arTonDelay[01](IN:=, PT:=T#1S , Q=> , ET=> );
arTonDelay[02](IN:= , PT:=T#1S , Q=> , ET=> );//注液延时使用
arTonDelay[03](IN:= , PT:=T#10S , Q=> , ET=> );
arTonDelay[04](IN:= , PT:=T#0.1S , Q=> , ET=> );
arTonDelay[05](IN:= , PT:=T#0.1S , Q=> , ET=> );
arTonDelay[06](IN:= , PT:=T#0.1S , Q=> , ET=> );
arTonDelay[07](IN:=NOT  fbXAxisMove.xbusy, PT:=T#0.1S , Q=> , ET=> );//TipAuto使用
arTonDelay[08](IN:=NOT  fbYAxisMove.xbusy , PT:=T#0.1S , Q=> , ET=> );//TipAuto使用
arTonDelay[09](IN:= NOT  fbZAxisMove.xbusy, PT:=T#0.1S , Q=> , ET=> );//TipAuto使用
arTonDelay[10](IN:= NOT fbStirAxis.xbusy, PT:=T#0.1S , Q=> , ET=> );//TipAuto使用
END_ACTION

ACTION FlowAuto:

//-----------------------------------------初始化是否完成判断----------------------------------------------
IF NOT station.xInitDone 
THEN
 	station.iStepAuto:=0;
 	station.xDone:=FALSE;
	station.xRunningOffProhibit := FALSE ;//运行中信号Off禁止
ELSIF station.xRunning OR  
(tsModuleProcess[bXCounter+1].xProcessStarted AND  NOT tsModuleProcess[bXCounter+1].xProcessCompleted)//注液流程
THEN
//-----------------------------------------动作步骤--------------------------------------------------------
CASE station.iStepAuto OF	  
	0: //----Home Step，等待启动----
		IF station.xDisabled 
			AND station.xCanRun 
			AND NOT fbMachine[1].xStopped 
			AND NOT station.xSingleRunning 
		THEN
			station.xDone:=TRUE;
		END_IF
		
		IF  station.xSingleRunning 
			OR station.xCanRun 
			AND NOT station.xDone 
			AND NOT station.xDisabled 
			AND NOT fbMachine[1].xStopped
		THEN
			station.xCycleEnable:=TRUE;
			station.xDone:= FALSE;  
			station.iStepAuto:= 10;
		END_IF
    10: //复位数据 
			FOR i:=1 TO gc_ModuleProNo BY 1 DO
				MEMSET(ADR(tsModuleProcess[i]),0,SIZEOF(tsModuleProcess[i]));
			END_FOR
			station.iStepAuto:=15;
	
	 15://程序分类选择
			IF NOT   fbMachine[1].xTryRun THEN
					 IF  station.xSingleRunning AND stCalibration.xNeedCalibration THEN//进入校准程序
							stCalibration.xWindowsTrigger:=TRUE;
							station.iStepAuto:=1000;
					 ELSE //进入正常程序
						 station.iStepAuto:=20;
					 END_IF
		 ELSE
					 station.iStepAuto:=20;
			END_IF
	20:////Restore_after_Estop_Process1 上载数据流程
			IF  station.xSingleRunning THEN  //OR fbMachine[1].xTryRun THEN
					station.iStepAuto :=45; 
			ELSIF tsModuleProcess[1].xProcessNotStarted AND NOT  tsModuleProcess[1].xProcessStarted THEN
					station.iStepAuto :=21; (*process not started*)
			ELSIF  tsModuleProcess[1].xProcessStarted AND NOT  tsModuleProcess[1].xProcessCompleted THEN
				 station.iStepAuto :=21 ;(*process started*)
			ELSIF  tsModuleProcess[1].xProcessCompleted AND NOT tsModuleProcess[1].xQDataCompleted  THEN
					station.iStepAuto :=30  ;(*process completed*)
			ELSIF tsModuleProcess[1].xQDataCompleted THEN
					station.iStepAuto :=30;(*Qdata completed *)
			ELSE
					station.iStepAuto :=21; 
			END_IF	
	21:	
			tsModuleProcess[1].xProcessNotStarted :=TRUE;
			station.iStepAuto :=25;
	25://数据load 
		tsModuleProcess[1].xProcessStarted:=TRUE;
		MEMCPY(ADR(arProcessDataStation[1]),ADR(arMainlineFixtureData[arCurFixtureNumStation[3]]),SIZEOF(arMainlineFixtureData[arCurFixtureNumStation[3]]));
		MEMCPY(ADR(arProcessDataStation[2]),ADR(arMainlineFixtureData[arCurFixtureNumStation[4]]),SIZEOF(arMainlineFixtureData[arCurFixtureNumStation[4]]));
		tsModuleProcess[1].xProcessCompleted:=TRUE;	
		tsModuleProcess[1].xQDataCompleted:=TRUE;	
		station.iStepAuto:= 30;
	/////产品流程开始	
	30: //判断产品状态
			 IF NOT  fbMachine[1].xTryRun THEN
					IF    station.xEmptyDone THEN //清料完成
							 station.iStepAuto:=998;
					ELSIF     //清料程序执行条件
							 arProcessDataStation[1].stProduct.xEmptying AND 
							 arProcessDataStation[2].stProduct.xEmptying AND 
							 NOT xSensorReached[1] AND  NOT   xSensorReached[2] THEN
										station.xEmptying :=TRUE;	
									  station.iStepAuto:= 2000; 
					ELSIF //第一站由于需要增加节拍增加了并行程序，所以写入请料的时机不好把控
					 			//在本站增加此条件以修正请料信号的位置
							 arProcessDataStation[1].stProduct.xEmptying AND 
							 arProcessDataStation[2].stProduct.xEmptying AND 
							  xSensorReached[1] AND  xSensorReached[2] THEN
										arProcessDataStation[1].stProduct.xEmptying :=FALSE; 		
								    arProcessDataStation[2].stProduct.xEmptying :=FALSE;
										arProcessDataStation[1].xMaterialOnOff :=TRUE; 		
								    arProcessDataStation[2].xMaterialOnOff :=TRUE;  
									  station.iStepAuto:= 40;
					ELSIF   (arProcessDataStation[1].xMaterialOnOff   AND
								  arProcessDataStation[2].xMaterialOnOff ) OR
									(xSensorReached[1] AND   xSensorReached[2])  THEN
										station.iStepAuto:= 40;  
					ELSIF		 NOT arProcessDataStation[1].xMaterialOnOff   AND
								   NOT arProcessDataStation[2].xMaterialOnOff  AND 
									 NOT xSensorReached[1]  AND  NOT xSensorReached[2]  THEN
									station.iStepAuto:= 998;
					END_IF
			 ELSE
					 station.iStepAuto:= 40;
			 END_IF
	40://写入NOK按钮
		IF   arManualNOKHmiButton[2]  AND NOT station.xSingleRunning THEN
			station.iStepAuto:=155;
			arManualNOKHmiButton[2]:=FALSE;
		ELSE
			 station.iStepAuto:=45;
		END_IF
	
	//////产品流程开始
	45://循环开始次数为1，总循环为2
			 bXCounter:=1;
	    station.iStepAuto:= 50;

	50:////Restore_after_Estop_Process1/2 注液流程1/2
			IF  station.xSingleRunning  OR fbMachine[1].xTryRun THEN
					station.iStepAuto :=80; 
			ELSIF tsModuleProcess[bXCounter+1].xProcessNotStarted AND NOT  tsModuleProcess[bXCounter+1].xProcessStarted THEN
					station.iStepAuto :=100; (*process not started*)
			ELSIF  tsModuleProcess[bXCounter+1].xProcessStarted AND NOT  tsModuleProcess[bXCounter+1].xProcessCompleted THEN
				 station.iStepAuto :=155 ;(*process started*)
			ELSIF  tsModuleProcess[bXCounter+1].xProcessCompleted AND NOT tsModuleProcess[bXCounter+1].xQDataCompleted  THEN
					station.iStepAuto :=150  ;(*process completed*)
			ELSIF tsModuleProcess[bXCounter+1].xQDataCompleted THEN
					station.iStepAuto :=160;(*Qdata completed *)
			ELSE
					station.iStepAuto :=80; 
			END_IF

	80://流程未开始
			 tsModuleProcess[bXCounter+1].xProcessNotStarted:=TRUE;
		 		station.iStepAuto:= 90;
	90://水平调整气缸伸出
		IF  iBoxChoose =1 THEN
			(*上层水平调整气缸*)
			fbHOZAdjustCyl_1.xAuto :=TRUE;
		//	fbHOZAdjustCyl_2.xAuto :=TRUE;
			IF  fbHOZAdjustCyl_1.xWP_Delay THEN// AND fbHOZAdjustCyl_2.xWP_Delay  THEN
					station.iStepAuto:= 100;
			END_IF
		ELSIF  iBoxChoose= 2 THEN
			(*下层水平调整气缸*)
			fbHOZAdjustCyl_3.xAuto :=TRUE;
			//fbHOZAdjustCyl_4.xAuto :=TRUE;
			IF  fbHOZAdjustCyl_3.xWP_Delay  THEN//AND fbHOZAdjustCyl_4.xWP_Delay  THEN
					station.iStepAuto:= 100;
			END_IF
		END_IF	 
	100://XY轴去注液位置1、2
			fbXAxisMove.xMoveAuto[bXCounter+1]:=TRUE;
			fbYAxisMove.xMoveAuto[bXCounter+1]:=TRUE;
			IF fbXAxisMove.xMoveInPos[bXCounter+1]  AND fbYAxisMove.xMoveInPos[bXCounter+1]  THEN
				station.iStepAuto:=110;	
			END_IF
	110:	//防滴液气缸伸出
		fbROTCyl.xAuto:=TRUE;
		IF fbROTCyl.xWP_Delay THEN
			station.iStepAuto:=120;	
		END_IF
	120://Z轴下降去注液位置
		   fbZAxisMove.xMoveAuto[2]:=TRUE;
		IF  fbZAxisMove.xMoveInPos[2] THEN
			station.iStepAuto:=125;
		END_IF
	125://屏蔽注液
			FOR i:=1 TO  12 BY 1 DO
					arxPushBusy[i]:=FALSE;
		 END_FOR
			IF   axBypassSignal[2] OR fbMachine[1].xTryRun THEN
				station.iStepAuto:=145;
			ELSE
				station.iStepAuto:=130;
			END_IF
	130://开始注液
		  tsModuleProcess[bXCounter+1].xProcessStarted:=TRUE;
		 FOR i:=1 TO  12 BY 1 DO
						fbEasyPumps[i].stDeviceOpe.xPush_Auto[1]:=TRUE;
						IF  fbEasyPumps[i].xQBusy THEN
						 		arxPushBusy[i]:=TRUE;
						END_IF
		 END_FOR
		 	FOR   i :=1 TO 12 BY  1  DO
			 			IF NOT  arxPushBusy[i] THEN
						 		EXIT;
						ELSIF i =12 THEN
						 	  station.iStepAuto:=140;	
					  END_IF
			END_FOR
	140://注液结束
					arTonDelay[02](IN:=FALSE );
					 IF   	fbEasyPumps[1].xQDone AND
									fbEasyPumps[2].xQDone AND
									fbEasyPumps[3].xQDone AND
								  fbEasyPumps[4].xQDone AND
									fbEasyPumps[5].xQDone AND
									fbEasyPumps[6].xQDone AND
									fbEasyPumps[7].xQDone AND
								  fbEasyPumps[8].xQDone AND
									fbEasyPumps[9].xQDone AND
									fbEasyPumps[10].xQDone AND
									fbEasyPumps[11].xQDone AND
								  fbEasyPumps[12].xQDone THEN						
								 station.iStepAuto:=145;	
					 END_IF
	145://注液完成
		tsModuleProcess[bXCounter+1].xProcessCompleted:=TRUE;
		 station.iStepAuto:=150;	
	150://写入结果
				arProcessDataStation[bXCounter].xMaterialOnOff:=TRUE;
				arProcessDataStation[bXCounter].stProduct.xlidInjecting_OK:=TRUE;
				arProcessDataStation[bXCounter].stProduct.xlidInjecting_NOK:=FALSE;	
			 tsModuleProcess[bXCounter].xQDataCompleted:=TRUE;
			 station.iStepAuto:=160;
	155://注液失败
				arProcessDataStation[bXCounter].xMaterialOnOff:=TRUE;
				arProcessDataStation[bXCounter].stProduct.xlidInjecting_OK:=FALSE;
				arProcessDataStation[bXCounter].stProduct.xlidInjecting_NOK:=TRUE;	
				station.iStepAuto:=160;
	160://Z轴上升
		  fbZAxisMove.xMoveAuto[1]:=TRUE;
		IF  fbZAxisMove.xMoveInPos[1] THEN
			station.iStepAuto:=170;
		END_IF
	170://防滴漏气缸收回
		fbROTCyl.xAuto:=FALSE;
		IF fbROTCyl.xHP_Delay THEN
			station.iStepAuto:=180;	
		END_IF
	180://循环+1
		 	bXCounter:=bXCounter +1 ;
			station.iStepAuto:=190;
	190://检查循环次数
			IF   bXCounter<=2 THEN
				station.iStepAuto:=50;
			ELSE
				station.iStepAuto:=200;
			END_IF
	200://水平调整气缸收回
			IF  iBoxChoose =1 THEN
			(*上层水平调整气缸*)
			fbHOZAdjustCyl_1.xAuto :=FALSE;
		//	fbHOZAdjustCyl_2.xAuto :=FALSE;
			IF  fbHOZAdjustCyl_1.xHP_Delay THEN  // AND fbHOZAdjustCyl_2.xHP_Delay  THEN
					station.iStepAuto:= 210;
			END_IF
		ELSIF  iBoxChoose= 2 THEN
			(*下层水平调整气缸*)
			fbHOZAdjustCyl_3.xAuto :=FALSE;
		//	fbHOZAdjustCyl_4.xAuto :=FALSE;
			IF  fbHOZAdjustCyl_3.xHP_Delay  THEN // AND fbHOZAdjustCyl_4.xHP_Delay  THEN
					station.iStepAuto:= 210;
			END_IF
		END_IF
	210:////产品流程结束	
		station.iStepAuto:= 220;
		
	220://Restore_after_Estop_Process4 数据传输 
			IF  station.xSingleRunning THEN // OR fbMachine[1].xTryRun THEN
					station.iStepAuto :=998; 
			ELSIF tsModuleProcess[4].xProcessNotStarted AND NOT  tsModuleProcess[4].xProcessStarted THEN
					station.iStepAuto :=550; (*process not started*)
			ELSIF  tsModuleProcess[4].xProcessStarted AND NOT  tsModuleProcess[4].xProcessCompleted THEN
				 station.iStepAuto :=550 ;(*process started*)
			ELSIF  tsModuleProcess[4].xProcessCompleted AND NOT tsModuleProcess[4].xQDataCompleted  THEN
					station.iStepAuto :=560  ;(*process completed*)
			ELSIF tsModuleProcess[4].xQDataCompleted THEN
					station.iStepAuto :=999;(*Qdata completed *)
			ELSE
					station.iStepAuto :=550; 
			END_IF
	550://数据unload
			tsModuleProcess[4].xProcessNotStarted :=TRUE;
			tsModuleProcess[4].xProcessStarted :=TRUE;
			MEMCPY(ADR(arMainlineFixtureData[arCurFixtureNumStation[3]]),ADR(arProcessDataStation[1]),SIZEOF(arProcessDataStation[1]));
			MEMCPY(ADR(arMainlineFixtureData[arCurFixtureNumStation[4]]),ADR(arProcessDataStation[2]),SIZEOF(arProcessDataStation[2]));
			station.iStepAuto:= 560;
		
	560:
			tsModuleProcess[4].xProcessCompleted :=TRUE;
			station.iStepAuto:= 570;
 	570://本地数据清除
			//MEMSET(ADR(arProcessDataStation[1]),0,SIZEOF(arProcessDataStation[1]));
			//MEMSET(ADR(arProcessDataStation[2]),0,SIZEOF(arProcessDataStation[2]));
			tsModuleProcess[4].xQDataCompleted:=TRUE;
			arManualNOKHmiButton[2]:=FALSE;
			station.iStepAuto:= 998;
		
	998://----Single Run Finish----
		station.iStepAuto :=999;
		IF NOT station.xSingleContinuousRun THEN
			station.xSingleRunFlag:=FALSE;
		END_IF
		station.xCycleEnable:=FALSE;	
		station.xDone:=TRUE;
		
	999://XY伺服回参考位置
			fbXAxisMove.xMoveAuto[1]:=TRUE;
			fbYAxisMove.xMoveAuto[1]:=TRUE;
			IF fbXAxisMove.xMoveInPos[1]  AND fbYAxisMove.xMoveInPos[1]  THEN
				station.iStepAuto:=0;	
			END_IF
	{region "蠕动泵校准程序"}
	1000://切换窗口
			stCalibration.xWindowsTrigger:=TRUE;
			iCalibStep:=station.iStepAuto;
			station.iStepAuto:=1010;
	1010://等待人工安装好校准工装,
		 stCalibration.strCalibHmi:='Please Load Calibration Tool and then press Start Button ';
		IF    stCalibration.xStartButtonHmi THEN
			station.iStepAuto:=1020;
		END_IF
			 	iCalibStep:=station.iStepAuto;
	1020://开始循环
		 	FOR i:=1 TO 12 BY 1 DO
				 IF 	NOT arxRudongPumpCalibBypass[i] THEN
						 stCalibration.iYCounter:=i;
						 EXIT;
				 END_IF
			END_FOR
			stCalibration.iXCounter:=1;
			//stCalibration.iYCounter:=1;
			iCalibStep:=station.iStepAuto;
			station.iStepAuto:=1030;
		{region "初始化开始"}	
	1030://初始化蠕动泵
			stCalibration.strCalibHmi:='All RuDongPump is initing，please Wait it';
			station.iStepAuto:=station.iStepAuto +1;
			iCalibStep:=station.iStepAuto;
	1031://蠕动泵初始化开始
				 FOR i:=1 TO  12 BY 1 DO
						fbEasyPumps[i].stDeviceOpe.xStop_auto:=TRUE;
						IF	NOT fbEasyPumps[i].xQBusy  THEN
								EXIT;
						ELSIF   i =12 THEN
									iCalibStep:=station.iStepAuto;
									station.iStepAuto:=station.iStepAuto +1;		
					 	END_IF						
				 END_FOR
	1032://蠕动泵停
					iCalibStep:=station.iStepAuto;
					IF   fbEasyPumps[1].xQDone AND 
							 fbEasyPumps[2].xQDone AND 
							 fbEasyPumps[3].xQDone AND 
							 fbEasyPumps[4].xQDone AND 
							 fbEasyPumps[5].xQDone AND 
							 fbEasyPumps[6].xQDone AND 
							 fbEasyPumps[7].xQDone AND 
							 fbEasyPumps[8].xQDone AND 
							 fbEasyPumps[9].xQDone AND 
							 fbEasyPumps[10].xQDone AND 
							 fbEasyPumps[11].xQDone AND
							 fbEasyPumps[12].xQDone THEN
							station.iStepAuto:=station.iStepAuto +1;
					END_IF
	1033://初始化称
					fbMCk.xIReset:=TRUE;
					iCalibStep:=station.iStepAuto;
				 station.iStepAuto:=station.iStepAuto +1;
	1034://等待初始化完成
					iCalibStep:=station.iStepAuto;
					IF fbMCk.xQRdyCmd THEN
						station.iStepAuto:=station.iStepAuto +1;
					END_IF
	1035://停止称的检测
					fbMCk.stDeviceOpe.xAcquireWeight_Stop_HMI:=TRUE;
					iCalibStep:=station.iStepAuto;
					station.iStepAuto:=station.iStepAuto +1;
	1036://等待完成
					IF fbMCk.xQRdyCmd THEN
							station.iStepAuto:=station.iStepAuto +1;
					END_IF	
						 	iCalibStep:=station.iStepAuto;
	1037://称清零
				iCalibStep:=station.iStepAuto;
				fbMCk.stDeviceOpe.xClearZeroInstanly_HMI:=TRUE;
				IF  fbMCK.xQBusy THEN
							station.iStepAuto:=station.iStepAuto +1;	
				END_IF
	1038://等待清零结束
				IF	fbMCk.xQDone THEN
						station.iStepAuto:=1040;
				END_IF		
					iCalibStep:=station.iStepAuto;	
{endregion}
	
{region "蠕动泵校准程序开始"}
	1040://计算XY轴移动目标位置
			stCalibration.strCalibHmi:='X\Y AXis move to Target Position，please Wait it';
			///机构还未调整好暂时屏蔽移动功能,后续开放出来
			stData.Axis[3].rMovePosition[6]:=fbXAxisMove.rMovePosition[4];//+(stCalibration.iXCounter -1)*9.0;
			stData.Axis[4].rMovePosition[6]:=fbYAxisMove.rMovePosition[4];//+(stCalibration.iYCounter -1)*9.0;
			iCalibStep:=station.iStepAuto;
			station.iStepAuto:=1045;
	1045://XY轴移动到位
				fbXAxisMove.xMoveAuto[6]:=TRUE;
				fbYAxisMove.xMoveAuto[6]:=TRUE;
			IF  fbXAxisMove.xMoveInPos[6]  AND fbYAxisMove.xMoveInPos[6] THEN
				station.iStepAuto:=1050;
			END_IF
			iCalibStep:=station.iStepAuto;
	1050://打开防滴液气缸
				fbROTCyl.xAuto:=TRUE;
				IF fbROTCyl.xWP_Delay THEN
					station.iStepAuto:=1060;	
				END_IF
				iCalibStep:=station.iStepAuto;
	1060://Z轴去校准位置
				fbZAxisMove.xMoveAuto[3]:=TRUE;
				IF  fbZAxisMove.xMoveInPos[3] THEN
					station.iStepAuto:=1069;
				END_IF
				iCalibStep:=station.iStepAuto;
							
	1069://注液次数设定
				 _InjectCounuter :=1 ;
				iCalibStep:=station.iStepAuto;				
				 station.iStepAuto:=station.iStepAuto +1 ;
	1070:
				stCalibration.strCalibHmi:='Auto Calibration is Running，please Wait it';
				iCalibStep:=station.iStepAuto;
				station.iStepAuto:=station.iStepAuto +1 ;	
				
	1071://等待校准就绪
				IF fbMCK.xQRdyCmd AND  fbEasyPumps[stCalibration.iYCounter].xQRdyCmd THEN 
						station.iStepAuto:=station.iStepAuto +1 ;	
				END_IF		
				iCalibStep:=station.iStepAuto;
	1072://秤体清零	
				fbMCK.stDeviceOpe.xClearZeroInstanly_Auto:=TRUE;
				IF  fbMCK.xQBusy THEN
						station.iStepAuto:=station.iStepAuto +1 ;		 
				END_IF
				iCalibStep:=station.iStepAuto;
				
	1073://清零完成
				IF fbMCK.xQDone THEN
				 		//stCalibration.rMckVolume:=fbMCK.stParOut.rCurrentWeight;
					 arrMckDisplay[_InjectCounuter]:=fbMCK.stParOut.rCurrentWeight;
					 stCalibration.rMckVolume:=fbMCK.stParOut.rCurrentWeight;
					iCalibStep:=station.iStepAuto;
					station.iStepAuto:=station.iStepAuto +1 ;		
				END_IF
	1074://等待稳定时间
				 tSteadyTimer(IN:=TRUE,PT:=T#1S);
				 IF tSteadyTimer.Q THEN
					 tSteadyTimer(IN:=FALSE);
					 station.iStepAuto:=1077;	
				 END_IF	
					iCalibStep:=station.iStepAuto;
	1077://蠕动泵校准地址
				stData.EasyPumps[stCalibration.iYCounter].iModuleAdress:=stCalibration.iXCounter;
				stCalibration.rRudongPumpVolume:= stData.EasyPumps[stCalibration.iYCounter].rCalFluVolume;;														
				stCalibration.iInjectCounter :=3;//默认注液次数
				 //密度计算公式，ρ＝m/V 
					IF stCalibration.iType=1 THEN
						stCalibration.rDensity:=1;
					ELSIF stCalibration.iType=2 THEN
						stCalibration.rDensity:=0.8;
					END_IF
					iCalibStep:=station.iStepAuto;
					station.iStepAuto:=station.iStepAuto +1 ;		
	1078://启动单通道注液
				iCalibStep:=station.iStepAuto;
				fbEasyPumps[stCalibration.iYCounter].stDeviceOpe.xModulePush_Auto:=TRUE;
				IF	fbEasyPumps[stCalibration.iYCounter].xQBusy  THEN
						 tSteadyTimer(IN:=FALSE);
						 station.iStepAuto:=station.iStepAuto +1 ;	
				END_IF
				
	1079://等待稳定时间
				iCalibStep:=station.iStepAuto;
				IF    fbEasyPumps[stCalibration.iYCounter].xQDone THEN
							 tSteadyTimer(IN:=TRUE,PT:=T#500MS);
							 IF tSteadyTimer.Q THEN
									 tSteadyTimer(IN:=FALSE);
									 station.iStepAuto:=station.iStepAuto +1 ;	
							 END_IF
				END_IF
	1080://获取称重稳态结果
					iCalibStep:=station.iStepAuto;
					fbMCK.stDeviceOpe.xAcquireWeight_Steady_Auto:=TRUE;
					IF  fbMCK.xQBusy THEN
						station.iStepAuto:=station.iStepAuto +1 ;	
					END_IF
					
	1081://等待完成
					 iCalibStep:=station.iStepAuto;
					 IF fbMCK.xQDone THEN
							 station.iStepAuto:=1084 ;	
					 END_IF	
	1084://获取称重结果
					iCalibStep:=station.iStepAuto;
					arrMckDisplay[_InjectCounuter]:=fbMCK.stParOut.rCurrentWeight/stCalibration.rDensity;
					station.iStepAuto:=station.iStepAuto +1 ;
					
	1085://判断是否相差太多
					iCalibStep:=station.iStepAuto;
					IF 	ABS (stCalibration.rRudongPumpVolume - arrMckDisplay[_InjectCounuter])>0.5*stCalibration.rRudongPumpVolume THEN
								station.iStepAuto:=1070 ;
					ELSE
							 station.iStepAuto:=station.iStepAuto +1 ;
					END_IF
					

	1086://检查蠕动泵注液次数
				iCalibStep:=station.iStepAuto;	
				IF   _InjectCounuter >= stCalibration.iInjectCounter THEN
				 			 _InjectCounuter:=1;
							 stCalibration.rMckVolume:=0.0;
							 station.iStepAuto:=station.iStepAuto +1 ;
							
				ELSE
							_InjectCounuter:=_InjectCounuter +1;
				 			station.iStepAuto:=1070;
				END_IF
				
	1087://三次注液后算出平均实际液量
				FOR  i:= 1 TO stCalibration.iInjectCounter BY 1 DO
				 		stCalibration.rMckVolume:= stCalibration.rMckVolume + arrMckDisplay[i];
				END_FOR
				stCalibration.rMckVolume:=stCalibration.rMckVolume/stCalibration.iInjectCounter;
				stData.EasyPumps[stCalibration.iYCounter].rModuleRealFluVolume:=stCalibration.rMckVolume;
				iCalibStep:=station.iStepAuto;
				station.iStepAuto:=station.iStepAuto +1 ;	
	1088://写入通道实际液量
				iCalibStep:=station.iStepAuto;
				fbEasyPumps[stCalibration.iYCounter].stDeviceOpe.xCalibAction_Auto:=TRUE;
				IF 	fbEasyPumps[stCalibration.iYCounter].xQBusy THEN
						station.iStepAuto:=station.iStepAuto +1 ;	
				END_IF
	1089://写入完成
					iCalibStep:=station.iStepAuto;
				 	IF 	fbEasyPumps[stCalibration.iYCounter].xQDone THEN
						station.iStepAuto:=station.iStepAuto +1 ;	
					END_IF
	1090://开始校准
				iCalibStep:=station.iStepAuto;
				fbEasyPumps[stCalibration.iYCounter].stDeviceOpe.xAdjust_Auto:=TRUE;
				IF 	fbEasyPumps[stCalibration.iYCounter].xQBusy THEN
						station.iStepAuto:=station.iStepAuto +1 ;	
				END_IF				
	1091://等待校准结束
				iCalibStep:=station.iStepAuto;
				IF NOT 	fbEasyPumps[stCalibration.iYCounter].xQBusy  THEN
					  IF NOT fbEasyPumps[stCalibration.iYCounter].xQDone   THEN
										 //校准了但是需要重新测试下
										 station.iStepAuto:=1040 ;		
						ELSE
									   station.iStepAuto:=station.iStepAuto +1;	
						END_IF
				END_IF			
	1092://Z轴回参考点
		//	fbZAxisMove.xMoveAuto[1]:=TRUE;
		//	IF   fbZAxisMove.xMoveInPos[1] THEN
			 		iCalibStep:=station.iStepAuto;
					 station.iStepAuto:=1095;
		//	END_IF
	1095://校准完成,移动到下一个位置
			stCalibration.iXCounter:=stCalibration.iXCounter +1;
			iCalibStep:=station.iStepAuto;
			station.iStepAuto:=1100;		
	1100://判断X轴循环 
			IF    stCalibration.iXCounter>8 THEN
						 IF stCalibration.iYCounter <12 THEN
									 FOR i:= (stCalibration.iYCounter+1) TO 12 BY 1 DO
													IF  NOT  arxRudongPumpCalibBypass[i] THEN
																stCalibration.iYCounter:= i;
																EXIT;
													END_IF
									 END_FOR
						 ELSIF stCalibration.iYCounter >=12 THEN
										stCalibration.iYCounter:=stCalibration.iYCounter+1;
						 END_IF
							stCalibration.iXCounter:=1;
							 station.iStepAuto:=1110;
			ELSE
					 station.iStepAuto:=1035;
			END_IF
			iCalibStep:=station.iStepAuto;
	1110://判断Y轴循环
			IF   stCalibration.iYCounter >12 THEN
					 stCalibration.iYCounter:=1;
					 stCalibration.iXCounter:=1;
					 station.iStepAuto:=1130;
			ELSE
					station.iStepAuto:=1120;
			END_IF
			iCalibStep:=station.iStepAuto;
	1120://等待下一组按钮按下
			stCalibration.strCalibHmi:='Wait Press Next Button HMI';
			IF stCalibration.xNextButtonHmi THEN
				station.iStepAuto:=1040;
			END_IF
			iCalibStep:=station.iStepAuto;
			
	1130://校准完成
			stCalibration.strCalibHmi:='Calibration Completed，wait press Completed button HMI';
			IF  stCalibration.xCompletedButtonHmi THEN
					 stCalibration.xNeedCalibration:=FALSE;	
					 station.iStepAuto:=1140;
			END_IF
			iCalibStep:=station.iStepAuto;
	1140://再按一次完成按钮关闭当前窗口
			stCalibration.strCalibHmi:='Close Current windows，wait press Completed button HMI';
			IF  stCalibration.xCompletedButtonHmi THEN
					 stCalibration.xWindowsTrigger:=FALSE;
					 station.iStepAuto:=1200;
			END_IF	
			iCalibStep:=station.iStepAuto;
	1200:///校准完成，请将工位初始化
		 iCalibStep:=station.iStepAuto;
			stCalibration.strCalibHmi:='Calibration Completed，Init station Now Please';
	1300://校准报错，请将工位初始化后继续
		 	 iCalibStep:=station.iStepAuto;
			 stCalibration.strCalibHmi:='Calibration Aborted，Init station Now Please';	 
	{endregion}		
	{region "清料程序"}	 
	2000://写入数据
		 	arProcessDataStation[1].xMaterialOnOff:=FALSE;
			arProcessDataStation[1].stProduct.xlidInjecting_OK:=FALSE;
			arProcessDataStation[1].stProduct.xlidInjecting_NOK:=FALSE;	
			arProcessDataStation[2].xMaterialOnOff:=FALSE;
			arProcessDataStation[2].stProduct.xlidInjecting_OK:=FALSE;
			arProcessDataStation[2].stProduct.xlidInjecting_NOK:=FALSE;	
			arProcessDataStation[1].stProduct.xEmptying:=TRUE;
			arProcessDataStation[2].stProduct.xEmptying:=TRUE;	
		 	MEMCPY(ADR(arMainlineFixtureData[arCurFixtureNumStation[3]]),ADR(arProcessDataStation[1]),SIZEOF(arProcessDataStation[1]));
			MEMCPY(ADR(arMainlineFixtureData[arCurFixtureNumStation[4]]),ADR(arProcessDataStation[2]),SIZEOF(arProcessDataStation[2]));
		 	station.iStepAuto:=2010;
	2010://允许主流线前进
		 			station.xDone:=TRUE;
				  station.iStepAuto:=2020;
  2020://停止蠕动泵
				FOR i:=1 TO gc_uiRudongPump BY 1 DO
					fbEasyPumps[i].stDeviceOpe.xStop_Auto:=TRUE;
				END_FOR
		   	station.iStepAuto :=2030;
	2030://等待蠕动泵全部停止
				IF   fbEasyPumps[1].xQDone AND 
							 fbEasyPumps[2].xQDone AND 
							 fbEasyPumps[3].xQDone AND 
							 fbEasyPumps[4].xQDone AND 
							 fbEasyPumps[5].xQDone AND 
							 fbEasyPumps[6].xQDone AND 
							 fbEasyPumps[7].xQDone AND 
							 fbEasyPumps[8].xQDone AND 
							 fbEasyPumps[9].xQDone AND 
							 fbEasyPumps[10].xQDone AND 
							 fbEasyPumps[11].xQDone AND
							 fbEasyPumps[12].xQDone THEN
							station.iStepAuto :=2040;
				END_IF
				
	2040://XYZ轴回参考位
				fbXAxisMove.xMoveAuto[1]:=TRUE;
				fbYAxisMove.xMoveAuto[1]:=TRUE;
				IF fbXAxisMove.xMoveInPos[1]  AND
				   fbYAxisMove.xMoveInPos[1]  THEN
					station.iStepAuto:=2100;	
				END_IF
	2100://当站清料完成
		 		station.xEmptying:=FALSE;
				station.xEmptyDone:=TRUE;
			  station.iStepAuto:=0;			 
	{endregion}
		 
		 
	ELSE
		;	
END_CASE
END_IF
{region "蠕动泵校准报警处理"}
//超时报警
	tCalibrationTimeOut(IN:= (iCalibStep = station.iStepAuto) AND iCalibStep >=1020 AND   iCalibStep <1120 , PT:=T#10S , Q=> , ET=> );
	//报警状态
		IF  fbMCK.xQError OR fbEasyPumps[stCalibration.iYCounter].xQError OR   tCalibrationTimeOut.Q THEN
					stCalibration.xError:=TRUE;		
					MEMSET(ADR(fbEasyPumps[stCalibration.iYCounter].stDeviceOpe),0,SIZEOF(fbEasyPumps[stCalibration.iYCounter].stDeviceOpe));
			 		MEMSET(ADR(fbMCK.stDeviceOpe),0,SIZEOF(fbMCK.stDeviceOpe));
					IF   stCalibration.xReset THEN
							fbMCK.xIReset:=TRUE;
							fbEasyPumps[stCalibration.iYCounter].xIReset:=TRUE;	 
							station.iStepAuto:=1300;
							stCalibration.xWindowsTrigger:=FALSE;
							iCalibStep:=0; 
					END_IF
		ELSE
					stCalibration.xError:=FALSE;		
		END_IF
//区分报警
	IF fbMCK.xQError THEN
				stCalibration.strCalibHmi:='Balance Error,Please check it';		
	ELSIF  fbRuDongPump[stCalibration.iYCounter].xError THEN
				stCalibration.strCalibHmi:='RudongPump Error,Please check it';	 
  ELSIF tCalibrationTimeOut.Q THEN
				stCalibration.strCalibHmi:='Calibration Timeout,Please check it'; 
	END_IF						 
{endregion}
END_ACTION

ACTION FlowInit:
IF NOT station.xIniting THEN
  station.iStepInit:=0;    
ELSE
//--------------------------------------------初始化步序----------------------------------
CASE station.iStepInit OF	
 0://  
 		iRudongPumpEmptyStep:=0;//复位排空流程
  	IF station.xIniting THEN	
  	  station.iStepInit:=10;	
  	END_IF	
10://复位数据
	FOR   i:=1 TO 12 BY 1	DO
	 	fbEasyPumps[i].xIReset:=TRUE;
		 arxPushBusy[i]:=FALSE;
	END_FOR
	fbMCK.xIReset:=TRUE;
	FOR i:=1 TO gc_ModuleProNo BY 1 DO
				MEMSET(ADR(tsModuleProcess[i]),0,SIZEOF(tsModuleProcess[i]));
	END_FOR
	station.iStepInit :=15;
15://伺服上电
   fbXAxisMove.xPowerInit := TRUE ;
	 fbYAxisMove.xPowerInit := TRUE ;
	 fbZAxisMove.xPowerInit := TRUE ;
	IF fbXAxisMove.xPowerOn AND   fbYAxisMove.xPowerOn AND  fbZAxisMove.xPowerOn THEN 
    	station.iStepInit:=20;	
	END_IF	
20://停止蠕动泵
		 FOR i:=1 TO  12 BY 1 DO
						fbEasyPumps[i].stDeviceOpe.xStop_Auto:=TRUE;
						IF  fbEasyPumps[i].xQBusy THEN
						 		arxPushBusy[i]:=TRUE;
						END_IF
		 END_FOR
		 	FOR   i :=1 TO 12 BY  1  DO
			 			IF NOT  arxPushBusy[i] THEN
						 		EXIT;
						ELSIF i =12 THEN
						 	  station.iStepInit:=25;	
					  END_IF
			END_FOR

25://等待蠕动泵全部停止
				 IF   		fbEasyPumps[1].xQDone AND
									fbEasyPumps[2].xQDone AND
									fbEasyPumps[3].xQDone AND
								  fbEasyPumps[4].xQDone AND
									fbEasyPumps[5].xQDone AND
									fbEasyPumps[6].xQDone AND
									fbEasyPumps[7].xQDone AND
								  fbEasyPumps[8].xQDone AND
									fbEasyPumps[9].xQDone AND
									fbEasyPumps[10].xQDone AND
									fbEasyPumps[11].xQDone AND
								  fbEasyPumps[12].xQDone THEN						
								 station.iStepInit:=30;	
					 END_IF;	
	
	
30://Z轴伺服上升
		fbZAxisMove.xMoveAuto[1]:=TRUE;
		IF fbZAxisMove.xMoveInPos[1]   THEN
			station.iStepInit:=40;	
		END_IF	
40://防滴液气缸回原
	fbROTCyl.xInit:=TRUE;
	IF fbROTCyl.xHP_Delay THEN
		station.iStepInit :=50;
	END_IF

50://XY轴回参考位
		fbXAxisMove.xMoveAuto[1]:=TRUE;
		fbYAxisMove.xMoveAuto[1]:=TRUE;
		IF fbXAxisMove.xMoveInPos[1]  AND fbYAxisMove.xMoveInPos[1]  THEN
			station.iStepInit:=90;	
		END_IF

90://水平调整气缸收回
	fbHOZAdjustCyl_1.xInit :=TRUE;
   // fbHOZAdjustCyl_2.xInit :=TRUE;
    fbHOZAdjustCyl_3.xInit :=TRUE;
   // fbHOZAdjustCyl_4.xInit :=TRUE;
	IF  fbHOZAdjustCyl_1.xHP_Delay AND 
	//	fbHOZAdjustCyl_2.xHP_Delay AND
		fbHOZAdjustCyl_3.xHP_Delay THEN
	//	fbHOZAdjustCyl_4.xHP_Delay THEN
		station.iStepInit:=100;	
	END_IF
	
100:
		station.iStepInit:=999;	
999://初始化完成	
	station.iStepInit:=0;
	station.xInitDone:=TRUE;  
END_CASE
END_IF
END_ACTION

ACTION General:
{region "清除过程记录"}
CASE bClearProcessStep OF
	0:	
		IF	 S08_MainLine.xClearProcessStatus THEN
			FOR i:=1 TO gc_ModuleProNo BY 1 DO
				MEMSET(ADR(tsModuleProcess[i]),0,SIZEOF(tsModuleProcess[i]));
			END_FOR
			bClearProcessStep:=10;
		END_IF
	10:
		xClearModuleProcessDone:=TRUE;
		bClearProcessStep:=20;
	20:
		IF NOT S08_MainLine.xClearProcessStatus THEN
			xClearModuleProcessDone:=FALSE;
			bClearProcessStep:=30;
		END_IF
	30:  
			bClearProcessStep:=0;
END_CASE
	 
{endregion}
	 
{region "蠕动泵排空"}
RudongPump_R_TRIG[1](CLK:=xAllRudongPumpEmpty , Q=> );
RudongPump_R_TRIG[2](CLK:=xRudongPumpEmptyDone , Q=> );
//超时报警
	tEmptyTimeOut(IN:= (iRudongPumpEmptyOldStep =iRudongPumpEmptyStep AND iRudongPumpEmptyStep <>0) , PT:=T#10S , Q=> , ET=> );
	IF		tEmptyTimeOut.Q THEN
				iRudongPumpEmptyStep:=0;
				station.adwAlarm[2].0	:=	TRUE	;//S02注液工位排空超时
	END_IF
CASE  iRudongPumpEmptyStep OF
		 0://等待触发信号
				 IF  RudongPump_R_TRIG[1].Q THEN
							iRudongPumpEmptyStep:= iRudongPumpEmptyStep +1;
				 ELSIF	RudongPump_R_TRIG[2].Q THEN
							iRudongPumpEmptyStep:=5;		 
				 END_IF
				
		 1://XY轴到排液位置
							iRudongPumpEmptyOldStep :=iRudongPumpEmptyStep;		
						 fbXAxisMove.xMoveAuto[5]:=TRUE;
						 fbYAxisMove.xMoveAuto[5]:=TRUE;
					 IF  fbXAxisMove.xMoveInPos[5]  AND fbYAxisMove.xMoveInPos[5] THEN
							iRudongPumpEmptyStep:= iRudongPumpEmptyStep +1;
					 END_IF		 
					  
		 2://防滴液气缸打开
						 	iRudongPumpEmptyOldStep :=iRudongPumpEmptyStep;
						 fbROTCyl.xAuto:=TRUE;
						 IF fbROTCyl.xWP_Delay THEN
								 iRudongPumpEmptyStep:= iRudongPumpEmptyStep +1;
						 END_IF
						 
		 3://Z轴去校准位置
						iRudongPumpEmptyOldStep :=iRudongPumpEmptyStep;
						 fbZAxisMove.xMoveAuto[4]:=TRUE;
						 IF  fbZAxisMove.xMoveInPos[4] THEN
							 iRudongPumpEmptyStep:= iRudongPumpEmptyStep +1;
						 END_IF
						
		 4://开始排空液体
						iRudongPumpEmptyOldStep :=iRudongPumpEmptyStep;	
						FOR i:=1 TO  12 BY 1 DO
							  IF   NOT  arxRudongPumpEmptyBypass[i] THEN
										fbEasyPumps[i].stDeviceOpe.xFullSpeedPush_Hmi:=TRUE;
								END_IF
									arxPushBusy[i]:=FALSE;
					 END_FOR
						
					  iRudongPumpEmptyStep:= 0;		
		 5://等待结束
						iRudongPumpEmptyOldStep :=iRudongPumpEmptyStep;	
						 FOR i:=1 TO  12 BY 1 DO
									 fbEasyPumps[i].stDeviceOpe.xFullSpeedStop_Hmi:=TRUE;	
									IF   	 fbEasyPumps[i].xQBusy THEN
												arxPushBusy[i]:=TRUE;
									END_IF		
						 END_FOR		
							 FOR i:=1 TO  12 BY 1 DO
									 	IF   NOT  	 arxPushBusy[i] THEN
												EXIT;
										ELSIF  i =12 THEN
												iRudongPumpEmptyStep:= iRudongPumpEmptyStep +1;		 
										END_IF			
							 END_FOR
		6://等待结束			
			 				iRudongPumpEmptyOldStep :=iRudongPumpEmptyStep;	
			 			 IF   fbEasyPumps[1].xQDone AND
									fbEasyPumps[2].xQDone AND
									fbEasyPumps[3].xQDone AND
								  fbEasyPumps[4].xQDone AND
									fbEasyPumps[5].xQDone AND
									fbEasyPumps[6].xQDone AND
									fbEasyPumps[7].xQDone AND
								  fbEasyPumps[8].xQDone AND
									fbEasyPumps[9].xQDone AND
									fbEasyPumps[10].xQDone AND
									fbEasyPumps[11].xQDone AND
								  fbEasyPumps[12].xQDone THEN						
								 iRudongPumpEmptyStep:= iRudongPumpEmptyStep +1;	
					 END_IF
		7://结束
							 iRudongPumpEmptyStep:= 0;		
END_CASE	
{endregion}
	 
{region "手动校准蠕动泵"}
IF  stManualCalib.xReset THEN
			  stManualCalib.xError:=FALSE;
			  stManualCalib.iOldMCalibStep:=0;
			  stManualCalib.iMCalibStep:=0;
			  stManualCalib.xBusy  :=FALSE;
			  stManualCalib.xDone :=FALSE;	  	 
			fbEasyPumps[stManualCalib.iPumpContorller].xIReset:=TRUE;
			fbMCK.xIReset:=TRUE;
END_IF
IF  NOT  stManualCalib.xBusy THEN
 		stManualCalib.xRdyCmd:=TRUE;
ELSE
 		stManualCalib.xRdyCmd:=FALSE;	
END_IF
tMCalibTimeOut(IN:= (stManualCalib.iMCalibStep =stManualCalib.iOldMCalibStep) AND stManualCalib.iMCalibStep<>0 , PT:= T#25S, Q=> , ET=> );
IF		tMCalibTimeOut.Q THEN
 	stManualCalib.xError:=TRUE;
	stManualCalib.iMCalibStep:=0;
END_IF
	 
			
				 
						
							 
//
//CASE stManualCalib.iMCalibStep OF
// 0://等待按键
//		IF  stManualCalib.xStart  AND
//			  stManualCalib.iPumpContorller>=1 AND 
//				stManualCalib.iPumpContorller<=12 AND 
//				stManualCalib.iPumpModule>=1 AND 
//				stManualCalib.iPumpModule<=9 THEN
//			  stManualCalib.xModulePushStart:=FALSE;		 
//				stManualCalib.xModulePushOK:=FALSE;			
//				stManualCalib.xCalibTestStart:=FALSE;				 
//				stManualCalib.xCalibTestOK:=FALSE;						
//				stManualCalib.xRecordDataStart:=FALSE;	
//				stManualCalib.xRecordDataOK:=FALSE;						 
//				stManualCalib.xStart  :=FALSE;
//				stManualCalib.xBusy  :=TRUE;
//				stManualCalib.xDone :=FALSE;	 
//				stManualCalib.iMCalibStep:=stManualCalib.iMCalibStep +1;
//		 END_IF
//1://参数赋值
//	 	stManualCalib.iOldMCalibStep:=stManualCalib.iMCalibStep;
//		stData.EasyPumps[stManualCalib.iPumpContorller].rCalFluVolume:=stManualCalib.rSetVolume;
//		stData.EasyPumps[stManualCalib.iPumpContorller].iModuleAdress:=stManualCalib.iPumpModule;
//		stData.EasyPumps[stManualCalib.iPumpContorller].rCalTime:=stManualCalib.rRunTime;
//		stData.EasyPumps[stManualCalib.iPumpContorller].rCalNum:=stManualCalib.iCycleNum;
//		stData.EasyPumps[stManualCalib.iPumpContorller].rModuleRealFluVolume:=stManualCalib.rAverageRealVolume;
//		stData.EasyPumps[stManualCalib.iPumpContorller].rCalBackAngle:=stManualCalib.iBackAngle;
//		stManualCalib.iMCalibStep:=stManualCalib.iMCalibStep +1;
//2://写入校准参数
//	 	stManualCalib.iOldMCalibStep:=stManualCalib.iMCalibStep;
//		stManualCalib.iMCalibStep:=stManualCalib.iMCalibStep +1;	
//3://等待写入完成
//	 	stManualCalib.iOldMCalibStep:=stManualCalib.iMCalibStep;
//	  stManualCalib.xModulePushStart:=TRUE;
//		stManualCalib.xModulePushOK:=FALSE;
//		stManualCalib.iMCalibStep:=stManualCalib.iMCalibStep +1;	
//4://清除原有数据
//	 	stManualCalib.iOldMCalibStep:=stManualCalib.iMCalibStep;
//		MEMSET(ADR(stManualCalib.arrRealVolume[1]),0,SIZEOF(stManualCalib.arrRealVolume));
//		stManualCalib.rAverageRealVolume:=0; 
//		stManualCalib.iInjectCounter:=1;
//	 	stManualCalib.iMCalibStep:=stManualCalib.iMCalibStep +1;	
//5://称清零
//	 	stManualCalib.iOldMCalibStep:=stManualCalib.iMCalibStep;
//		IF  stManualCalib.iInjectCounter >1 AND  stManualCalib.xRepeatMode THEN
//				//如果需要连续注液，不需要中间清零
//				stManualCalib.iMCalibStep:=stManualCalib.iMCalibStep +2;	
//		ELSE
//				 fbMCK.stDeviceOpe.xClearZeroInstanly_HMI:=TRUE;
//				 IF fbMCK.xQBusy THEN
//							 stManualCalib.iMCalibStep:=stManualCalib.iMCalibStep +1;	
//					END_IF
//		END_IF
//6://等待清零完成
//	 	stManualCalib.iOldMCalibStep:=stManualCalib.iMCalibStep;
//	  IF  fbMCK.xQDone THEN
//			  	stManualCalib.iMCalibStep:=stManualCalib.iMCalibStep +1;
//		 ELSIF  fbMCK.xQError THEN
//				  fbMCK.xIReset:=TRUE;
//					stManualCalib.iMCalibStep:=5;	
//		 END_IF
//7://开始单通道注液
//	 	stManualCalib.iOldMCalibStep:=stManualCalib.iMCalibStep;
//	  fbEasyPumps[stManualCalib.iPumpContorller].stDeviceOpe.xModulePush_Auto:=TRUE;
//		IF  fbEasyPumps[stManualCalib.iPumpContorller].xQBusy THEN
//				stManualCalib.iMCalibStep:=stManualCalib.iMCalibStep +1;	
//		END_IF
//8://等待注液完成
//	 	stManualCalib.iOldMCalibStep:=stManualCalib.iMCalibStep;
//	 	stManualCalib.tStableDelay(IN:= FALSE);
//	 	IF  fbEasyPumps[stManualCalib.iPumpContorller].xQDone THEN
//				stManualCalib.iMCalibStep:=stManualCalib.iMCalibStep +1;	
//		END_IF
//9://等待
//	 IF (( stManualCalib.xModulePushStart AND stManualCalib.xRepeatMode AND  stManualCalib.iInjectCounter =5)OR
//			stManualCalib.xCalibTestStart OR
//			stManualCalib.xRecordDataStart) OR
//			  NOT  stManualCalib.xRepeatMode  THEN
//				
//					 stManualCalib.tStableDelay(IN:= TRUE, PT:=T#6S , Q=> , ET=> );
//					 IF  stManualCalib.tStableDelay.Q THEN
//									stManualCalib.tStableDelay(IN:= FALSE);
//									stManualCalib.iMCalibStep:=stManualCalib.iMCalibStep +1;	
//					 END_IF			 
//	 ELSE
//			 //如果需要连续注液，只有在最后一次才需要注液
//						stManualCalib.iMCalibStep:=stManualCalib.iMCalibStep +2;	
//	 END_IF
//10://读取称的读数
//	 	stManualCalib.iOldMCalibStep:=stManualCalib.iMCalibStep;
//	 	fbMCK.stDeviceOpe.xAcquireWeight_RealTime_HMI:=TRUE;
//		IF fbMCK.xQBusy THEN
//					stManualCalib.iMCalibStep:=stManualCalib.iMCalibStep +1;	
//		END_IF
//11://等待完成
//	 	stManualCalib.iOldMCalibStep:=stManualCalib.iMCalibStep;
//	  IF  fbMCK.xQDone THEN
//				IF  (fbMCK.stParOut.rCurrentWeight <=stManualCalib.rSetVolume*0.1 AND NOT stManualCalib.xRepeatMode)  THEN
//										stManualCalib.iMCalibStep:=5;
//				ELSE
//							IF  stManualCalib.xModulePushStart   THEN
//									stManualCalib.arrRealVolume[stManualCalib.iInjectCounter]:=fbMCK.stParOut.rCurrentWeight;
//							ELSIF  stManualCalib.xCalibTestStart THEN
//								 stManualCalib.arrRealVolume[stManualCalib.iCalibCounter]:=fbMCK.stParOut.rCurrentWeight;	
//							ELSIF  stManualCalib.xRecordDataStart THEN
//									stManualCalib.arrRecordVolume[stManualCalib.iRecordCounter]:=fbMCK.stParOut.rCurrentWeight;
//							END_IF
//			  			stManualCalib.iMCalibStep:=stManualCalib.iMCalibStep +1;	
//					END_IF
//		 ELSIF  fbMCK.xQError THEN
//				  fbMCK.xIReset:=TRUE;
//					 stManualCalib.iMCalibStep:=5;
//		 END_IF
//12://注液计数
//	 	stManualCalib.iOldMCalibStep:=stManualCalib.iMCalibStep;
//	 	IF  stManualCalib.xModulePushStart THEN
//	  			stManualCalib.iInjectCounter := stManualCalib.iInjectCounter +1;
//		ELSIF   stManualCalib.xCalibTestStart THEN
//				 	stManualCalib.iCalibCounter := stManualCalib.iCalibCounter +1;
//		ELSIF  stManualCalib.xRecordDataStart THEN
//						stManualCalib.iRecordCounter := stManualCalib.iRecordCounter +1;
//		END_IF
//	 	stManualCalib.iMCalibStep:=stManualCalib.iMCalibStep +1;	
//13://
//	 	stManualCalib.iOldMCalibStep:=stManualCalib.iMCalibStep;
//	 	IF   stManualCalib.xModulePushStart THEN
//				IF 	 stManualCalib.iInjectCounter >5 THEN
//							stManualCalib.iMCalibStep:=stManualCalib.iMCalibStep +1;
//				ELSE
//							stManualCalib.iMCalibStep:=5;
//				END_IF
//		ELSIF   stManualCalib.xCalibTestStart THEN
//				IF 	 stManualCalib.iCalibCounter >5 THEN
//							stManualCalib.iMCalibStep:=stManualCalib.iMCalibStep +1;
//				ELSE
//							stManualCalib.iMCalibStep:=5;
//				END_IF
//		ELSIF   stManualCalib.xRecordDataStart THEN
//				IF 	 stManualCalib.iRecordCounter >50 THEN
//							stManualCalib.iMCalibStep:=stManualCalib.iMCalibStep +1;
//				ELSE
//							stManualCalib.iMCalibStep:=5;
//				END_IF			 
//		END_IF
//			 
//14://计算平均液量或者校准的精度
//	 	stManualCalib.iOldMCalibStep:=stManualCalib.iMCalibStep;
//		IF  stManualCalib.xModulePushStart THEN
//				   IF  NOT stManualCalib.xRepeatMode THEN
//								 FOR i:=1 TO 5 BY 1 DO
//											 stManualCalib.rAverageRealVolume:=stManualCalib.rAverageRealVolume +stManualCalib.arrRealVolume[i];
//								 END_FOR
//									stManualCalib.rAverageRealVolume:=stManualCalib.rAverageRealVolume/5;
//						ELSE
//									stManualCalib.rAverageRealVolume:=stManualCalib.arrRealVolume[5]/5; 
//						END_IF
//						stManualCalib.xModulePushStart:=FALSE;
//						stManualCalib.xModulePushOK:=TRUE;
//						stManualCalib.iMCalibStep:=stManualCalib.iMCalibStep +1;
//		 ELSIF  stManualCalib.xCalibTestStart THEN
//									stManualCalib.rESVolume:=FC_BubbleSort_Max(i_i_Counter:=5 , i_arrReal:= stManualCalib.arrRealVolume);//最大值
//									stManualCalib.rEIVolume:=FC_BubbleSort_Min(i_i_Counter:=5, i_arrReal:= stManualCalib.arrRealVolume);//最小值
//									stManualCalib.rESVolume:=(stManualCalib.rESVolume-stManualCalib.rSetVolume)/stManualCalib.rSetVolume;//上偏差
//									stManualCalib.rEIVolume:=(stManualCalib.rEIVolume-stManualCalib.rSetVolume)/stManualCalib.rSetVolume;//下偏差	 
//									 IF  stManualCalib.rESVolume>stData.EasyPumps[stManualCalib.iPumpContorller].iAccuracySet  OR 
//											 	stManualCalib.rEIVolume<-1*stData.EasyPumps[stManualCalib.iPumpContorller].iAccuracySet 	THEN
//											//-	>stData.EasyPumps[stManualCalib.iPumpContorller].iAccuracySet*0.5
//													 	FOR i:=1 TO 5 BY 1 DO
//																stManualCalib.rAverageRealVolume:=stManualCalib.rAverageRealVolume +stManualCalib.arrRealVolume[i];
//														END_FOR
//														 stManualCalib.rAverageRealVolume:=stManualCalib.rAverageRealVolume/5;
//													 stManualCalib.xCalibTestStart:=FALSE;
//													 stManualCalib.xCalibTestOK:=FALSE;
//												//如果上下偏差不均衡  我们需要进行微调处理
//										   IF  ABS(ABS( stManualCalib.rESVolume)-ABS(stManualCalib.rEIVolume))<=stData.EasyPumps[stManualCalib.iPumpContorller].iAccuracySet*0.5 THEN
//													 stManualCalib.iMCalibStep:=stManualCalib.iMCalibStep +1;
//											 ELSE
//													  stManualCalib.iMCalibStep:=stManualCalib.iMCalibStep +3;
//											 END_IF
//									 ELSE
//													 stManualCalib.xCalibTestStart:=FALSE;
//													 stManualCalib.xCalibTestOK:=TRUE;
//													 stManualCalib.xRecordDataStart:=TRUE;
//													 stManualCalib.xRecordDataOK:=FALSE;
//													 stManualCalib.iRecordCounter:=1;
//													 stManualCalib.iMCalibStep:=4;
//									 END_IF
//			ELSIF stManualCalib.xRecordDataStart THEN
//											stManualCalib.xRecordDataStart:=FALSE;
//											stManualCalib.xRecordDataOK:=TRUE;	
//											 stManualCalib.xBusy  :=FALSE;
//											 stManualCalib.xDone  :=TRUE;	 
//											 stManualCalib.iMCalibStep:=0;			
//		  END_IF
//15://写入校准参数
//	 	stManualCalib.iOldMCalibStep:=stManualCalib.iMCalibStep;
//				stData.EasyPumps[stManualCalib.iPumpContorller].rModuleRealFluVolume:=stManualCalib.rAverageRealVolume;
//				fbEasyPumps[stManualCalib.iPumpContorller].stDeviceOpe.xCalibAction_Hmi:=TRUE;
//				IF  fbEasyPumps[stManualCalib.iPumpContorller].xQBusy THEN
//							stManualCalib.iMCalibStep:=stManualCalib.iMCalibStep +1;	
//				END_IF
//16://等待写入完成
//	 	stManualCalib.iOldMCalibStep:=stManualCalib.iMCalibStep;
//	 	IF  fbEasyPumps[stManualCalib.iPumpContorller].xQDone THEN
//				stManualCalib.xCalibTestStart:=TRUE;
//				stManualCalib.iCalibCounter:=1;
//					stManualCalib.iMCalibStep:=20;	
//		END_IF	
//	
//17://开始微调
//	 	stManualCalib.iOldMCalibStep:=stManualCalib.iMCalibStep;
//		fbEasyPumps[stManualCalib.iPumpContorller].stDeviceOpe.xAdjust_Hmi:=TRUE;
//		IF  fbEasyPumps[stManualCalib.iPumpContorller].xQBusy THEN
//				stManualCalib.iMCalibStep:=stManualCalib.iMCalibStep +1;	
//		END_IF
//18://等待写入完成
//	 	stManualCalib.iOldMCalibStep:=stManualCalib.iMCalibStep;
//	 	IF  fbEasyPumps[stManualCalib.iPumpContorller].xQDone THEN
//				stManualCalib.iMCalibStep:=20;	
//		END_IF
//20://校准结束,开始测试校准效果
//			stManualCalib.iMCalibStep:=4;	 
 
//END_CASE
	//复位校准参数
IF  stManualCalib.iMCalibStep =0 THEN
			IF  stManualCalib.xInitCalibration THEN
					 	fbEasyPumps[stManualCalib.iPumpContorller].stDeviceOpe.xCalibInit_Auto:=TRUE;
						stManualCalib.xInitCalibration:=FALSE;
			END_IF
END_IF
{endregion}
{region "将记录的数据放入Excel中"}
Tc2_System.MEMCPY(ADR(arrVBARecordData),ADR(stManualCalib.arrRecordVolume),SIZEOF(stManualCalib.arrRecordVolume));
iEasyPumpController:= stManualCalib.iPumpContorller;
iEasyPumpGHead:=stManualCalib.iPumpModule;
iCycleCounter:=stManualCalib.iCycleNum;
rAccuracySet:=stData.EasyPumps[stManualCalib.iPumpContorller].iAccuracySet;
rSetVolume:=stManualCalib.rSetVolume;
rRunTime:=stManualCalib.rRunTime;
iBackAngle:=stManualCalib.iBackAngle;
iPumpType:=stData.EasyPumps[stManualCalib.iPumpContorller].iPumpType;
iSoftType:=stData.EasyPumps[stManualCalib.iPumpContorller].iHosePipeTypeSet;
iPumpHeadType:=stData.EasyPumps[stManualCalib.iPumpContorller].iPumpTypeSet;	 
{endregion}
{region '压力传感器循环读取'}

//循环触发
CASE  iRepeatLoadCellStep OF 
0://读取
	 IF  fbMachine[1].xAutoMode OR TRUE THEN
			 FOR i:=1 TO gc_uiLoadcellNum DO
						fbLoadCell[i].stDeviceOpe.xReadGROSSAuto:=TRUE;
						IF   fbLoadCell[i].xQBusy THEN
						 		arxLoadCellBusy[i]:=TRUE;
						END_IF
			 END_FOR
				FOR   i :=1 TO gc_uiLoadcellNum BY  1  DO
			 			IF NOT  arxLoadCellBusy[i] THEN
						 		EXIT;
						ELSIF i =gc_uiLoadcellNum THEN
						 	  iRepeatLoadCellStep:=iRepeatLoadCellStep +1;	
					  END_IF
			END_FOR
	 END_IF 
	1:	//等待
		 	iOldRepeatLoadCellStep :=iRepeatLoadCellStep;
			IF  fbLoadCell[1].xQDone AND 
					fbLoadCell[2].xQDone AND 
					fbLoadCell[3].xQDone AND 
					fbLoadCell[4].xQDone AND 
					fbLoadCell[5].xQDone AND 
					fbLoadCell[6].xQDone THEN
					 iRepeatLoadCellStep:=iRepeatLoadCellStep +1;	
			END_IF
	2://比较压力传感器的数值
		 	iOldRepeatLoadCellStep :=iRepeatLoadCellStep;	
			 FOR i:=1 TO gc_uiLoadcellNum DO
					IF  fbLoadCell[i].stParOut.rGROSSWeight< -100 THEN
							iRepeatLoadCellStep:=iRepeatLoadCellStep +1;	
							EXIT;	
					ELSIF  i=gc_uiLoadcellNum THEN
							iRepeatLoadCellStep:=iRepeatLoadCellStep +2;	
					END_IF
			 END_FOR
 3://数值异常
			IF    fbLoadCell[1].stParOut.rGROSSWeight<-100 THEN
								station.adwAlarm[2].01	:=	TRUE	;//	S02注液工位1号桶液量不足，请更换母液
			ELSIF    fbLoadCell[2].stParOut.rGROSSWeight< -100  THEN
								station.adwAlarm[2].02	:=	TRUE	;//	S02注液工位2号桶液量不足，请更换母液
			ELSIF    fbLoadCell[3].stParOut.rGROSSWeight< -100  THEN
								station.adwAlarm[2].03	:=	TRUE	;//	S02注液工位3号桶液量不足，请更换母液
			ELSIF    fbLoadCell[4].stParOut.rGROSSWeight< -100  THEN
								station.adwAlarm[2].04	:=	TRUE	;//	S02注液工位4号桶液量不足，请更换母液
			ELSIF    fbLoadCell[5].stParOut.rGROSSWeight< -100 THEN
								station.adwAlarm[2].05	:=	TRUE	;//	S02注液工位5号桶液量不足，请更换母液
			ELSIF    fbLoadCell[6].stParOut.rGROSSWeight< -100 THEN
								station.adwAlarm[2].06	:=	TRUE	;//	S02注液工位6号桶液量不足，请更换母液
			END_IF
			 
 4://数值正常,继续延时
			iOldRepeatLoadCellStep :=iRepeatLoadCellStep;
			tLoadCellDelay(IN:=TRUE , PT:=T#1S , Q=> , ET=> );
			IF  tLoadCellDelay.Q  THEN
			   		iRepeatLoadCellStep:=0;	
			END_IF
END_CASE
	 tLoadCellTimeout(IN:=  	iOldRepeatLoadCellStep =iRepeatLoadCellStep AND  iRepeatLoadCellStep<>0, PT:=T#10S , Q=> , ET=> );
IF  		tLoadCellTimeout.Q THEN
					station.adwAlarm[2].07	:=	TRUE	;//	S02注液工位压力传感器读取超时报警，请检查
END_IF
IF  fbMachine[1].xReset THEN
		iRepeatLoadCellStep:=0;
END_IF
				 
						
{endregion}
END_ACTION

ACTION ILC:

//---------------------------------------------------工站可执行-------------------------------------------------------
station.xCanRun :=TRUE ;

//---------------------------------------------------气缸动作条件-------------------------------------------
fbHOZAdjustCyl_1.xOffILC	:=	TRUE	;
fbHOZAdjustCyl_1.xOnILC	:=	TRUE	;
//fbHOZAdjustCyl_2.xOffILC	:=	TRUE	;
//fbHOZAdjustCyl_2.xOnILC	:=	TRUE	;
fbHOZAdjustCyl_3.xOffILC	:=	TRUE	;
fbHOZAdjustCyl_3.xOnILC	:=	TRUE	;
//fbHOZAdjustCyl_4.xOffILC	:=	TRUE	;
//fbHOZAdjustCyl_4.xOnILC	:=	TRUE	;
fbROTCyl.xOffILC	:=	TRUE	;
fbROTCyl.xOnILC	:=	TRUE;

//---------------------------------------------------伺服动作条件-------------------------------------------
fbXAxisMove.xRunILC := 					
fbXAxisMove.xMoveILC[1] :=					
fbxAxisMove.xMoveILC[2] :=					
fbxAxisMove.xMoveILC[3] :=					
fbxAxisMove.xMoveILC[4] :=					
fbxAxisMove.xMoveILC[5] := 		fbROTCyl.xHP_Sensor ;
fbYAxisMove.xRunILC := 			
fbYAxisMove.xMoveILC[1] :=					
fbYAxisMove.xMoveILC[2] :=					
fbYAxisMove.xMoveILC[3] :=					
fbYAxisMove.xMoveILC[4] :=					
fbYAxisMove.xMoveILC[5] := 	fbROTCyl.xHP_Sensor		 ;
fbZAxisMove.xRunILC := 	 				
fbZAxisMove.xMoveILC[1] :=					
fbZAxisMove.xMoveILC[2] :=					
fbZAxisMove.xMoveILC[3] :=					
fbZAxisMove.xMoveILC[4] :=					
fbZAxisMove.xMoveILC[5] := 		fbROTCyl.xWP_Sensor		;
fbStirAxis.xRunILC := 					
fbStirAxis.xMoveILC[1] :=					
fbStirAxis.xMoveILC[2] :=					
fbStirAxis.xMoveILC[3] :=					
fbStirAxis.xMoveILC[4] :=					
fbStirAxis.xMoveILC[5] := 		TRUE			;
///蠕动泵
fbEasyPumps[1].xideviceRunning:=
fbEasyPumps[2].xideviceRunning:=
fbEasyPumps[3].xideviceRunning:=
fbEasyPumps[4].xideviceRunning:=
fbEasyPumps[5].xideviceRunning:=
fbEasyPumps[6].xideviceRunning:=
fbEasyPumps[7].xideviceRunning:=
fbEasyPumps[8].xideviceRunning:=
fbEasyPumps[9].xideviceRunning:=
fbEasyPumps[10].xideviceRunning:=
fbEasyPumps[11].xideviceRunning:=
fbEasyPumps[12].xideviceRunning:=TRUE;


fbRudongPump[1].xDeviceRunning:=
fbRudongPump[2].xDeviceRunning:=
fbRudongPump[3].xDeviceRunning:=
fbRudongPump[4].xDeviceRunning:=
fbRudongPump[5].xDeviceRunning:=
fbRudongPump[6].xDeviceRunning:=
fbRudongPump[7].xDeviceRunning:=
fbRudongPump[8].xDeviceRunning:=
fbRudongPump[9].xDeviceRunning:=
fbRudongPump[10].xDeviceRunning:=
fbRudongPump[11].xDeviceRunning:=
fbRudongPump[12].xDeviceRunning:=TRUE;
//称
fbMCK.xIDeviceRunning:=TRUE;

fbAutoCal.xDeviceRunning:=TRUE;
END_ACTION

ACTION TipAuto:

//------------------------------------------------AutoTip Cylinder--------------------------------
station.adwAutoTip[1].00	:=	fbHOZAdjustCyl_1.xAutoTip	;
//station.adwAutoTip[1].01	:=	fbHOZAdjustCyl_2.xAutoTip	;
station.adwAutoTip[1].02	:=	fbHOZAdjustCyl_3.xAutoTip	;
//station.adwAutoTip[1].03	:=	fbHOZAdjustCyl_4.xAutoTip	;
station.adwAutoTip[1].04	:=	fbROTCyl.xAutoTip	;

//------------------------------------------------AutoTip Servo--------------------------------
//**************************************
FOR i:= 1 TO 5 BY 1 DO 
	IF fbXAxisMove.xMoveAuto[i] THEN
		fbXAxisMove.iPosNumber := i ;
	END_IF
	IF fbYAxisMove.xMoveAuto[i] THEN
		fbYAxisMove.iPosNumber := i ;
	END_IF
	IF fbZAxisMove.xMoveAuto[i] THEN
		fbZAxisMove.iPosNumber := i ;
	END_IF
	IF fbStirAxis.xMoveAuto[i] THEN
		fbStirAxis.iPosNumber := i ;
	END_IF
END_FOR


IF  fbMachine[1].xAutoMode AND NOT fbMachine[1].xRunning AND arTonDelay[7].Q  THEN
		IF fbXAxisMove.iPosNumber=1 AND NOT fbXAxisMove.xMoveInPos[1] THEN station.adwAutoTip[1].10:=TRUE; END_IF//轴伺服自动时位置不在位置1	
		IF fbXAxisMove.iPosNumber=2 AND NOT fbXAxisMove.xMoveInPos[2] THEN station.adwAutoTip[1].11:=TRUE; END_IF//轴伺服自动时位置不在位置2	
		IF fbXAxisMove.iPosNumber=3 AND NOT fbXAxisMove.xMoveInPos[3] THEN station.adwAutoTip[1].12:=TRUE; END_IF//轴伺服自动时位置不在位置3	
		IF fbXAxisMove.iPosNumber=4 AND NOT fbXAxisMove.xMoveInPos[4] THEN station.adwAutoTip[1].13:=TRUE; END_IF//轴伺服自动时位置不在位置4	
		IF fbXAxisMove.iPosNumber=5 AND NOT fbXAxisMove.xMoveInPos[5] THEN station.adwAutoTip[1].14:=TRUE; END_IF//轴伺服自动时位置不在位置5	
END_IF		
IF  fbMachine[1].xAutoMode AND NOT fbMachine[1].xRunning AND arTonDelay[8].Q  THEN		
		IF fbYAxisMove.iPosNumber=1 AND NOT fbYAxisMove.xMoveInPos[1] THEN station.adwAutoTip[1].15:=TRUE; END_IF//轴伺服自动时位置不在位置1	
		IF fbYAxisMove.iPosNumber=2 AND NOT fbYAxisMove.xMoveInPos[2] THEN station.adwAutoTip[1].16:=TRUE; END_IF//轴伺服自动时位置不在位置2	
		IF fbYAxisMove.iPosNumber=3 AND NOT fbYAxisMove.xMoveInPos[3] THEN station.adwAutoTip[1].17:=TRUE; END_IF//轴伺服自动时位置不在位置3	
		IF fbYAxisMove.iPosNumber=4 AND NOT fbYAxisMove.xMoveInPos[4] THEN station.adwAutoTip[1].18:=TRUE; END_IF//轴伺服自动时位置不在位置4	
		IF fbYAxisMove.iPosNumber=5 AND NOT fbYAxisMove.xMoveInPos[5] THEN station.adwAutoTip[1].19:=TRUE; END_IF//轴伺服自动时位置不在位置5	
END_IF	
IF  fbMachine[1].xAutoMode AND NOT fbMachine[1].xRunning AND arTonDelay[9].Q  THEN	
		IF fbZAxisMove.iPosNumber=1 AND NOT fbZAxisMove.xMoveInPos[1] THEN station.adwAutoTip[1].20:=TRUE; END_IF//轴伺服自动时位置不在位置1	
		IF fbZAxisMove.iPosNumber=2 AND NOT fbZAxisMove.xMoveInPos[2] THEN station.adwAutoTip[1].21:=TRUE; END_IF//轴伺服自动时位置不在位置2	
		IF fbZAxisMove.iPosNumber=3 AND NOT fbZAxisMove.xMoveInPos[3] THEN station.adwAutoTip[1].22:=TRUE; END_IF//轴伺服自动时位置不在位置3	
		IF fbZAxisMove.iPosNumber=4 AND NOT fbZAxisMove.xMoveInPos[4] THEN station.adwAutoTip[1].23:=TRUE; END_IF//轴伺服自动时位置不在位置4	
		IF fbZAxisMove.iPosNumber=5 AND NOT fbZAxisMove.xMoveInPos[5] THEN station.adwAutoTip[1].24:=TRUE; END_IF//轴伺服自动时位置不在位置5	
END_IF
IF  fbMachine[1].xAutoMode AND NOT fbMachine[1].xRunning AND arTonDelay[10].Q  THEN		
		IF fbStirAxis.iPosNumber=1 AND NOT fbStirAxis.xMoveInPos[1] THEN station.adwAutoTip[1].25:=TRUE; END_IF//轴伺服自动时位置不在位置1	
		IF fbStirAxis.iPosNumber=2 AND NOT fbStirAxis.xMoveInPos[2] THEN station.adwAutoTip[1].26:=TRUE; END_IF//轴伺服自动时位置不在位置2	
		IF fbStirAxis.iPosNumber=3 AND NOT fbStirAxis.xMoveInPos[3] THEN station.adwAutoTip[1].27:=TRUE; END_IF//轴伺服自动时位置不在位置3	
		IF fbStirAxis.iPosNumber=4 AND NOT fbStirAxis.xMoveInPos[4] THEN station.adwAutoTip[1].28:=TRUE; END_IF//轴伺服自动时位置不在位置4	
		IF fbStirAxis.iPosNumber=5 AND NOT fbStirAxis.xMoveInPos[5] THEN station.adwAutoTip[1].29:=TRUE; END_IF//轴伺服自动时位置不在位置5	
END_IF
END_ACTION

ACTION TipManual:
//--------------------------------------------ManualTip------------------------------------------------------

//-------------------------------------------气缸提示---------------------------------------------------------




/////////////////////////////////////////////////////////////////////////////////////////////////////////////////
END_ACTION

ACTION Z_Output:
(**************************气缸输出********************************)
QxS02HOZAdjustCyl_1WP	:=	fbHOZAdjustCyl_1.xWP_Valve	;
QxS02HOZAdjustCyl_1HP	:=	fbHOZAdjustCyl_1.xHP_Valve	;

QxS02HOZAdjustCyl_3WP	:=	fbHOZAdjustCyl_3.xWP_Valve	;
QxS02HOZAdjustCyl_3HP	:=	fbHOZAdjustCyl_3.xHP_Valve	;

QxS02ROTCylWP	:=	fbROTCyl.xWP_Valve	;
QxS02ROTCylHP	:=	fbROTCyl.xHP_Valve	;
END_ACTION

END_PROGRAM

// ---- POUs/003_FB/53_RudongPump/08_PeristalticPumpFB/梅特勒托利多秤/FB_MT_MKC.TcPOU
{attribute 'tc_no_symbol'}
FUNCTION_BLOCK FB_MT_MKC//METTLER电子秤
VAR_INPUT
	xExecute: BOOL;//指令执行
	xAbort: BOOL;//指令中断
	xEstop	:BOOL;//急停
	xDeviceRunning:BOOL;
	xResetRequest: BOOL;//复位操作
	stDeviceOpe	:ST_DeviceOpe;//秤体操作
	stpar		:ST_MCK_ParIn;
	stSysPar	:ST_SysPar;
	dwTimeOut: DWORD;//[ms],0 => no executing time limit	  
	xManualHMIControl : BOOL;
	xAutoMode    : BOOL;//0:mannal 1:auto
	xIniting     : BOOL;//初始化过程中  
END_VAR
VAR_OUTPUT
	xDone			: BOOL;(*完成条件满足*)
	xBusy			: BOOL;(*动作正在执行*)
	xError			: BOOL;(*错误条件满足*)
	eErrorID		: MT_MCK_ERROR;(*错误码*)
	eTCPErrorID 	:UDINT;(*TCPIP Client错误码*)
	xRdyCmd 		: BOOL;//代表指令准备完成
 	xRefOk          : BOOL;//初始化完成
	stParOut		: ST_MCK_ParOut;//参数输出
END_VAR

VAR
{attribute 'tc_no_symbol'}
	eState: STATE;//当前状态
{attribute 'tc_no_symbol'}
	xAborted: BOOL;(*指令被打断，一般是处于急停中*)
{attribute 'tc_no_symbol'}
	sFromServer			: T_MaxString := '';//(*string from server*)
{attribute 'tc_no_symbol'}
	rxBuffer			: ARRAY[1..MAX_PLCPRJ_RXBUFFER_SIZE] OF BYTE;//接收缓存区域(byte数组)
{attribute 'tc_no_symbol'}
	xFirstInvocation: BOOL := TRUE;	 
{attribute 'tc_no_symbol'}
	xTimeOut: BOOL;
{attribute 'tc_no_symbol'}
	tOperationTimer : TON;
{attribute 'tc_no_symbol'}
	_tDelay : TON;
{attribute 'tc_no_symbol'}
	_fbTcpIpClient	: FB_TcpIpClient;
{attribute 'tc_no_symbol'}
  	_first : BOOL;
{attribute 'tc_no_symbol'}
	_sReceiveData : T_MaxString := '';//实际发送和接收的数据
{attribute 'tc_no_symbol'}
	_sSendData : T_MaxString := '';//实际发送和接收的数据
{attribute 'tc_no_symbol'}
	_sReadDataTemp : T_MaxString := '';//实际发送和接收的数据
{attribute 'tc_no_symbol'}
	_iSendNGCount: INT;//发送NG计数。读取NG计数，读取数据计数
{attribute 'tc_no_symbol'}
	_iNGCount,_iReadNGCount: INT;// 
{attribute 'tc_no_symbol'}
	_iReadDataCount: INT;//发送NG计数。读取NG计数，读取数据计数 
{attribute 'tc_no_symbol'}	
	 _iStatusIndex: INT;//发送NG计数。读取NG计数，读取数据计数 
{attribute 'tc_no_symbol'}
	_iReadDataFristIndex : INT;
{attribute 'tc_no_symbol'}
	 _iReadDataLastIndex : INT;
{attribute 'tc_no_symbol'}
	_rHMIControl : R_TRIG;
{attribute 'tc_no_symbol'}
	_rManual : R_TRIG;
{attribute 'tc_no_symbol'}
	_fManual : F_TRIG;
{attribute 'tc_no_symbol'}
	_xModeChange : BOOL;
{attribute 'tc_no_symbol'}
	_diCmdState 	: DINT; 
{attribute 'tc_no_symbol'}
	_tonTimeout: TON;	
{attribute 'tc_no_symbol'}	
	_tonCmdTimeout: TON;	
{attribute 'tc_no_symbol'}	
	_tonDelay: TON;	
{attribute 'tc_no_symbol'}		
	_rOperaTrig	:ARRAY [1..15] OF R_TRIG;
{attribute 'tc_no_symbol'}
	eCmd:MT_MCK_CMD;
{attribute 'tc_no_symbol'}
	xAutomodeFlag:BOOL;
{attribute 'tc_no_symbol'}
	rTareSet		:REAL;
{attribute 'tc_no_symbol'}
	_rStopCmdTrig :R_TRIG;
{attribute 'tc_no_symbol'}
	_Stemp		:ARRAY [1..20] OF STRING;	
{attribute 'tc_no_symbol'}
	_xHMIOpe :BOOL;//是否有手动操作，是否有自动操作	
{attribute 'tc_no_symbol'}	
	 _xAutoOpe : BOOL;//是否有手动操作，是否有自动操作
{attribute 'tc_no_symbol'}		 
	 _xDone:BOOL;
{attribute 'tc_no_symbol'}	 
	 _rInit:R_TRIG;
END_VAR
VAR_TEMP
{attribute 'tc_no_symbol'}
	xAgain: BOOL;
END_VAR


IF NOT _first 
THEN
	_first := TRUE;
	_fbTcpIpClient.nRemotePort := stSysPar.nRemotePort;//端口号
	_fbTcpIpClient.sRemoteHost := stSysPar.sRemoteHost;//IP地址
ELSE
  xAgain:=0;
  _fbTcpIpClient();
	eTCPErrorID := _fbTcpIpClient.udiErrorID;
	xRdyCmd := eState = STATE.DORMANT AND eERRORID = MT_MCK_ERROR.No_ERROR;//检测是否允许指令控制(初始状态，没有报警发生)	
	xDone:=_xDone AND xExecute;
  _rInit(CLK:= xIniting);//检测是否是初始化中，如果是的去切换模式
  IF _rInit.Q
  THEN
   eState := STATE.RESETING;
  END_IF 	
	//检测是否有模式变化
_fManual(CLK:=xAutoMode);
_rManual(CLK:=xAutoMode);

IF eState <> STATE.DORMANT//只有在运行的时候，才会检测是否有模式切换发生
THEN
	IF _fManual.Q OR _rManual.Q
	THEN
		_xModeChange := TRUE;
	END_IF
END_IF
	//_fbTcpIpClient.xNeedReceive := xNeedReceive;//设置发送之后是否需要反馈信息
	REPEAT
		CASE eState OF
			STATE.DORMANT:
				HandleDormantState(xAgain=> xAgain);
			STATE.EXECUTING:
				HandleExecutingState(xAgain=> xAgain);
			STATE.DONE:
				HandleDoneState(xAgain=> xAgain);
			STATE.INERROR:
				HandleErrorState(xAgain=> xAgain);
			STATE.ABORTING:
				HandleAbortingState(xAgain=> xAgain);
			STATE.ABORTED:
				HandleAbortedState(xAgain=> xAgain);
			STATE.RESETING:
				HandleResettingState(xAgain=> xAgain);
			END_CASE
	UNTIL (xAgain=0)
	END_REPEAT
END_IF


//报错内容输出
CASE eErrorID OF 
	MT_MCK_ERROR.FLT_CMD_TIMEOUT:
		stParOut.sErrorID:='MT_MCK_ERROR.FLT_CMD_TIMEOUT';
	MT_MCK_ERROR.FLT_CmdFeedback:
		stParOut.sErrorID:='MT_MCK_ERROR.FLT_CmdFeedback';
	MT_MCK_ERROR.FLT_CommandCantSend:
		stParOut.sErrorID:='MT_MCK_ERROR.FLT_CommandCantSend';
	MT_MCK_ERROR.FLT_CONNECT:
		stParOut.sErrorID:='MT_MCK_ERROR.FLT_CONNECT';
	MT_MCK_ERROR.FLT_LogicaL:
		stParOut.sErrorID:='MT_MCK_ERROR.FLT_LogicaL';
	MT_MCK_ERROR.FLT_Par:
		stParOut.sErrorID:='MT_MCK_ERROR.FLT_Par';
	MT_MCK_ERROR.FLT_PARA:
		stParOut.sErrorID:='MT_MCK_ERROR.FLT_PARA';
	MT_MCK_ERROR.FLT_RDYCMD:
		stParOut.sErrorID:='MT_MCK_ERROR.FLT_RDYCMD';
	MT_MCK_ERROR.FLT_STOP_TIMEOUT:
		stParOut.sErrorID:='MT_MCK_ERROR.FLT_STOP_TIMEOUT';
	MT_MCK_ERROR.FLT_Syntax:
		stParOut.sErrorID:='MT_MCK_ERROR.FLT_Syntax';
	MT_MCK_ERROR.FLT_TOverMax:
		stParOut.sErrorID:='MT_MCK_ERROR.FLT_TOverMax';
	MT_MCK_ERROR.FLT_TOverMin:
		stParOut.sErrorID:='MT_MCK_ERROR.FLT_TOverMin';
	MT_MCK_ERROR.FLT_ZI:
		stParOut.sErrorID:='MT_MCK_ERROR.FLT_ZI';
	MT_MCK_ERROR.FLT_ZOverMax:
		stParOut.sErrorID:='MT_MCK_ERROR.FLT_ZOverMax';
	MT_MCK_ERROR.FLT_ZOverMin:
		stParOut.sErrorID:='MT_MCK_ERROR.FLT_ZOverMin';
	MT_MCK_ERROR.No_ERROR:
		stParOut.sErrorID:='MT_MCK_ERROR.No_ERROR';		
END_CASE


//手动自动操作检测
_xHMIOpe :=
			stDeviceOpe.xAcquireWeight_Continuous_HMI OR 
			stDeviceOpe.xAcquireWeight_RealTime_HMI OR 
			stDeviceOpe.xAcquireWeight_Steady_HMI OR 		
			stDeviceOpe.xAcquireWeight_Stop_HMI OR 					
			stDeviceOpe.xClearZero_HMI OR 
			stDeviceOpe.xClearZeroInstanly_HMI OR 
			stDeviceOpe.xlearTare_HMI OR 
			stDeviceOpe.xReadSerialNum_HMI OR 
			stDeviceOpe.xRestart_HMI OR 			
			stDeviceOpe.xSetTare_HMI 	OR
			stDeviceOpe.xShelling_HMI OR 	
			stDeviceOpe.xShellingInstanly_HMI;		
			
_xAutoOpe:=	
			stDeviceOpe.xAcquireWeight_Continuous_Auto OR 
			stDeviceOpe.xAcquireWeight_RealTime_Auto OR 
			stDeviceOpe.xAcquireWeight_Steady_Auto OR 		
			stDeviceOpe.xAcquireWeight_Stop_Auto OR 					
			stDeviceOpe.xClearZero_Auto OR 
			stDeviceOpe.xClearZeroInstanly_Auto OR 
			stDeviceOpe.xlearTare_Auto OR 
			stDeviceOpe.xReadSerialNum_Auto OR 
			stDeviceOpe.xRestart_Auto OR 			
			stDeviceOpe.xSetTare_Auto 	OR
			stDeviceOpe.xShelling_Auto OR 	
			stDeviceOpe.xShellingInstanly_Auto;

{attribute 'tc_no_symbol'}
METHOD PROTECTED AbortAction
VAR_INPUT
END_VAR
VAR_OUTPUT
	xComplete: BOOL;
	eErrorID: MT_MCK_ERROR;
END_VAR
(*
* Cleaning
* => abort all running operation
* => if an NBS.ERROR codition is reached, set eErrorID to a Value rather then NBS.ERROR.NO_ERROR 
*)
xComplete:=1;
eErrorID:=MT_MCK_ERROR.NO_ERROR;
END_METHOD

{attribute 'tc_no_symbol'}
METHOD PROTECTED CmdAcquireWeight_Continuous
VAR_OUTPUT
	xComplete: BOOL;
END_VAR
// return the real actual fault number
IF eERRORID <> MT_MCK_ERROR.No_ERROR
THEN
  RETURN;  
END_IF

CASE _diCmdState OF	
		
		
	0://清空发送与接收缓冲区
		_tonDelay(IN:= TRUE,pt:=T#1MS);//保证执行的是最新的一次
		stParOut.rWeightMax:=0;
		stParOut.rWeightMin:=0;
		SysMemSet( ADR( _sSendData ), 0, SIZEOF(_sSendData) );//清除发送区域
		SysMemSet( ADR( _sReadDataTemp ), 0, SIZEOF(_sReadDataTemp) );//清除接收报告数据缓存区域
		SysMemSet( ADR( sFromServer ), 0, SIZEOF(sFromServer) );//清除发送区域
		_fbTcpIpClient.xNeedReceive := TRUE;//默认都是需要有收发交互的		
		IF _tonDelay.Q THEN
			_tonDelay(IN:= FALSE,pt:=T#20MS);
			_diCmdState:=_diCmdState+1;	
		END_IF		
		
	1://拼接读取指令
		_tonDelay(IN:= _fbTcpIpClient.xRdyCmd ,pt:=T#1MS);
		_tonCmdTimeout(IN:= FALSE,pt:=T#2S);
		_sSendData := 'SI$R$N';
		IF _tonDelay.Q THEN 
			_tonDelay(IN:= FALSE,pt:=T#20MS);
			_fbTcpIpClient.xEnable := FALSE;
			_diCmdState:=_diCmdState+1;		
		END_IF		
		
	2://发送指令,等待接收成功
		_tonCmdTimeout(IN:=TRUE ,pt:=T#2S);
		SysMemCpy(ADR(_fbTcpIpClient.aToServer),ADR(_sSendData),SIZEOF(_sSendData));	
		_fbTcpIpClient.udiSendNumber := LEN(_sSendData);			
		_fbTcpIpClient.xEnable := TRUE;	
		IF _fbTcpIpClient.xDone//接收成功
		THEN			
			_fbTcpIpClient.xEnable := FALSE;
			sFromServer := _sReceiveData := _fbTcpIpClient.sFromServer;//传递接收数据		
			rxBuffer := _fbTcpIpClient.rxBuffer;		
			IF FIND(_sReceiveData,'$R$N') <> 0 AND FIND(_sReceiveData,'S') <>0			
			THEN
				IF FIND(_sReceiveData,'mg') <> 0 THEN
					_Stemp[1]:=RIGHT(_sReceiveData,LEN(_sReceiveData)-5);
					_Stemp[2]:=LEFT(_Stemp[1],FIND(_Stemp[1],'mg$R$N')-1);
					stParOut.rCurrentWeight := TO_REAL(_Stemp[2]);
					stParOut.sWeightUnit:='mg';				
				ELSE 
					IF FIND(_sReceiveData,'g') <> 0 THEN
						_Stemp[1]:=RIGHT(_sReceiveData,LEN(_sReceiveData)-5);
						_Stemp[2]:=LEFT(_Stemp[1],FIND(_Stemp[1],'g$R$N')-1);
						stParOut.rCurrentWeight := TO_REAL(_Stemp[2]);
						stParOut.sWeightUnit:='g';				
					END_IF				
				END_IF
				IF stParOut.rCurrentWeight>stParOut.rWeightMax THEN
					stParOut.rWeightMax:=stParOut.rCurrentWeight;
				END_IF
				IF stParOut.rCurrentWeight<stParOut.rWeightMin THEN
					stParOut.rWeightMin:=stParOut.rCurrentWeight;
				END_IF	
				_diCmdState:=_diCmdState+1;
			ELSIF FIND(_sReceiveData,'EL') <>0 THEN
				eErrorID:=MT_MCK_ERROR.FLT_LogicaL;//逻辑错误
				_diCmdState:=999;
			ELSIF FIND(_sReceiveData,'ES') <>0 THEN
				eErrorID:=MT_MCK_ERROR.FLT_Syntax;//语法错误
				_diCmdState:=999;				
			ELSIF FIND(_sReceiveData,'I') <>0 THEN
				eErrorID:=MT_MCK_ERROR.FLT_CommandCantSend;//指令条件不满足,无法发送
				_diCmdState:=999;				
			ELSIF FIND(_sReceiveData,'L') <>0 THEN
				eErrorID:=MT_MCK_ERROR.FLT_PARA;//参数错误
				_diCmdState:=999;				
			END_IF
		END_IF
		IF _tonCmdTimeout.Q THEN
			eErrorID:=MT_MCK_ERROR.FLT_CMD_TIMEOUT;
			_diCmdState:=999;
		END_IF
	
	3://判断是否停止读取	
			_diCmdState:=_diCmdState+1;
		
	4://
		xComplete := TRUE; 
		
	ELSE
		;	
END_CASE
END_METHOD

{attribute 'tc_no_symbol'}
METHOD PROTECTED CmdAcquireWeight_RealTime
VAR_OUTPUT
	xComplete: BOOL;
END_VAR
// return the real actual fault number
IF eERRORID <> MT_MCK_ERROR.No_ERROR
THEN
  RETURN;  
END_IF

CASE _diCmdState OF	
		
		
	0://清空发送与接收缓冲区
		_tonDelay(IN:= TRUE,pt:=T#1MS);//保证执行的是最新的一次
		SysMemSet( ADR( _Stemp ), 0, SIZEOF(_Stemp) );//清除缓存数据处理区域
		SysMemSet( ADR( _sSendData ), 0, SIZEOF(_sSendData) );//清除发送区域
		SysMemSet( ADR( _sReadDataTemp ), 0, SIZEOF(_sReadDataTemp) );//清除接收报告数据缓存区域
		SysMemSet( ADR( sFromServer ), 0, SIZEOF(sFromServer) );//清除发送区域
		_fbTcpIpClient.xNeedReceive := TRUE;//默认都是需要有收发交互的		
		IF _tonDelay.Q THEN
			_tonDelay(IN:= FALSE,pt:=T#20MS);
			_diCmdState:=_diCmdState+1;	
		END_IF		
		
	1://拼接读取指令
		_tonDelay(IN:= _fbTcpIpClient.xRdyCmd ,pt:=T#1MS);
		_tonCmdTimeout(IN:= FALSE,pt:=T#2S);
		_sSendData := 'SI$R$N';
		IF _tonDelay.Q THEN 
			_tonDelay(IN:= FALSE,pt:=T#20MS);
			_fbTcpIpClient.xEnable := FALSE;
			_diCmdState:=_diCmdState+1;		
		END_IF		
		
	2://发送指令,等待接收成功
		_tonCmdTimeout(IN:=TRUE ,pt:=T#2S);
		SysMemCpy(ADR(_fbTcpIpClient.aToServer),ADR(_sSendData),SIZEOF(_sSendData));	
		_fbTcpIpClient.udiSendNumber := LEN(_sSendData);			
		_fbTcpIpClient.xEnable := TRUE;	
		IF _fbTcpIpClient.xDone//接收成功
		THEN			
			_fbTcpIpClient.xEnable := FALSE;
			sFromServer := _sReceiveData := _fbTcpIpClient.sFromServer;//传递接收数据		
			rxBuffer := _fbTcpIpClient.rxBuffer;		
			IF FIND(_sReceiveData,'$R$N') <> 0 AND FIND(_sReceiveData,'S') <>0			
			THEN
				IF FIND(_sReceiveData,'mg') <> 0 THEN
					_Stemp[1]:=RIGHT(_sReceiveData,LEN(_sReceiveData)-5);
					_Stemp[2]:=LEFT(_Stemp[1],FIND(_Stemp[1],'mg$R$N')-1);
					stParOut.rCurrentWeight := TO_REAL(_Stemp[2]);
					stParOut.sWeightUnit:='mg';
				ELSE 
					IF FIND(_sReceiveData,'g') <> 0 THEN
						_Stemp[1]:=RIGHT(_sReceiveData,LEN(_sReceiveData)-5);
						_Stemp[2]:=LEFT(_Stemp[1],FIND(_Stemp[1],'g$R$N')-1);
						stParOut.rCurrentWeight := TO_REAL(_Stemp[2]);
						stParOut.sWeightUnit:='g';				
					END_IF				
				END_IF
				_diCmdState:=_diCmdState+1;
			ELSIF FIND(_sReceiveData,'EL') <>0 THEN
				eErrorID:=MT_MCK_ERROR.FLT_LogicaL;//逻辑错误
				_diCmdState:=999;
			ELSIF FIND(_sReceiveData,'ES') <>0 THEN
				eErrorID:=MT_MCK_ERROR.FLT_Syntax;//语法错误
				_diCmdState:=999;				
			ELSIF FIND(_sReceiveData,'I') <>0 THEN
				eErrorID:=MT_MCK_ERROR.FLT_CommandCantSend;//指令条件不满足,无法发送
				_diCmdState:=999;				
			ELSIF FIND(_sReceiveData,'L') <>0 THEN
				eErrorID:=MT_MCK_ERROR.FLT_PARA;//参数错误
				_diCmdState:=999;				
			END_IF
		END_IF
		IF _tonCmdTimeout.Q THEN
			eErrorID:=MT_MCK_ERROR.FLT_CMD_TIMEOUT;
			_diCmdState:=999;
		END_IF
	
	3://
		xComplete := TRUE; 
		
	ELSE
		;	
END_CASE
END_METHOD

{attribute 'tc_no_symbol'}
METHOD PROTECTED CmdAcquireWeight_Stop
VAR_OUTPUT
	xComplete: BOOL;
END_VAR
// return the real actual fault number
IF eERRORID <> MT_MCK_ERROR.No_ERROR
THEN
  RETURN;  
END_IF

CASE _diCmdState OF	
		
		
	0://清空发送与接收缓冲区
		_tonDelay(IN:= TRUE,pt:=T#20MS);//保证执行的是最新的一次
		SysMemSet( ADR( _Stemp ), 0, SIZEOF(_Stemp) );//清除缓存数据处理区域
		SysMemSet( ADR( _sSendData ), 0, SIZEOF(_sSendData) );//清除发送区域
		SysMemSet( ADR( _sReadDataTemp ), 0, SIZEOF(_sReadDataTemp) );//清除接收报告数据缓存区域
		SysMemSet( ADR( sFromServer ), 0, SIZEOF(sFromServer) );//清除发送区域
		_fbTcpIpClient.xNeedReceive := TRUE;//默认都是需要有收发交互的		
		IF _tonDelay.Q THEN
			_tonDelay(IN:= FALSE,pt:=T#20MS);
			_diCmdState:=_diCmdState+1;	
		END_IF		
		
	1://拼接读取指令
		_tonDelay(IN:= _fbTcpIpClient.xRdyCmd ,pt:=T#10MS);
		_tonCmdTimeout(IN:= FALSE,pt:=T#2S);
		_sSendData := 'SI$R$N';
		IF _tonDelay.Q THEN 
			_tonDelay(IN:= FALSE,pt:=T#20MS);
			_fbTcpIpClient.xEnable := FALSE;
			_diCmdState:=_diCmdState+1;		
		END_IF		
		
	2://发送指令,等待接收成功
		SysMemCpy(ADR(_fbTcpIpClient.aToServer),ADR(_sSendData),SIZEOF(_sSendData));	
		_fbTcpIpClient.udiSendNumber := LEN(_sSendData);				
		_fbTcpIpClient.xEnable := TRUE;	
		IF _fbTcpIpClient.xDone//接收成功
		THEN			
			_fbTcpIpClient.xEnable := FALSE;
			sFromServer := _sReceiveData := _fbTcpIpClient.sFromServer;//传递接收数据		
			rxBuffer := _fbTcpIpClient.rxBuffer;		
			IF FIND(_sReceiveData,'$R$N') <> 0 AND FIND(_sReceiveData,'S') <> 0						
			THEN
				_Stemp[1]:=RIGHT(_sReceiveData,LEN(_sReceiveData)-4);
				_Stemp[2]:=LEFT(_Stemp[1],FIND(_Stemp[1],'g$R$N')-1);
				stParOut.rCurrentWeight := TO_REAL(_Stemp[2]);
				_diCmdState:=_diCmdState+1;	
			END_IF
		END_IF
	
	3://
		xComplete := TRUE; 
		
	ELSE
		;	
END_CASE
END_METHOD

METHOD PROTECTED CmdClearTare
VAR_OUTPUT
	xComplete: BOOL;
END_VAR
// return the real actual fault number
IF eERRORID <> MT_MCK_ERROR.No_ERROR
THEN
  RETURN;  
END_IF

CASE _diCmdState OF	
		
		
	0://清空发送与接收缓冲区
		_tonDelay(IN:= TRUE,pt:=T#1MS);//保证执行的是最新的一次
		sysMEMSET( ADR( _Stemp ), 0, SIZEOF(_Stemp) );//清除缓存数据处理区域
		sysMEMSET( ADR( _sSendData ), 0, SIZEOF(_sSendData) );//清除发送区域
		sysMEMSET( ADR( _sReadDataTemp ), 0, SIZEOF(_sReadDataTemp) );//清除接收报告数据缓存区域
		sysMEMSET( ADR( sFromServer ), 0, SIZEOF(sFromServer) );//清除发送区域
		_fbTcpIpClient.xNeedReceive := TRUE;//默认都是需要有收发交互的		
		IF _tonDelay.Q THEN
			_tonDelay(IN:= FALSE,pt:=T#20MS);
			_diCmdState:=_diCmdState+1;	
		END_IF		
		
	1://拼接读取指令
		_tonDelay(IN:= _fbTcpIpClient.xRdyCmd ,pt:=T#1MS);
		_tonCmdTimeout(IN:= FALSE,pt:=T#2S);
		_sSendData := 'TAC$R$N';//清除皮重
		IF _tonDelay.Q THEN 
			_tonDelay(IN:= FALSE,pt:=T#20MS);
			_fbTcpIpClient.xEnable := FALSE;
			_diCmdState:=_diCmdState+1;		
		END_IF				
		
	2://发送指令,等待接收成功
		sysMEMCPY(ADR(_fbTcpIpClient.aToServer),ADR(_sSendData),SIZEOF(_sSendData));	
		_fbTcpIpClient.udiSendNumber := LEN(_sSendData);				
		_fbTcpIpClient.xEnable := TRUE;	
		IF _fbTcpIpClient.xDone//接收成功
		THEN			
			_fbTcpIpClient.xEnable := FALSE;
			sFromServer := _sReceiveData := _fbTcpIpClient.sFromServer;//传递接收数据		
			rxBuffer := _fbTcpIpClient.rxBuffer;		
			IF FIND(_sReceiveData,'$R$N') <> 0 AND FIND(_sReceiveData,'TAC') <> 0						
			THEN
				stParOut.rCurrentTareWight:=0;
				_diCmdState:=_diCmdState+1;
			ELSIF FIND(_sReceiveData,'EL') <>0 THEN
				eErrorID:=MT_MCK_ERROR.FLT_LogicaL;//逻辑错误
				_diCmdState:=999;
			ELSIF FIND(_sReceiveData,'ES') <>0 THEN
				eErrorID:=MT_MCK_ERROR.FLT_Syntax;//语法错误
				_diCmdState:=999;				
			ELSIF FIND(_sReceiveData,'I') <>0 THEN
				eErrorID:=MT_MCK_ERROR.FLT_CommandCantSend;//指令条件不满足,无法发送
				_diCmdState:=999;				
			ELSIF FIND(_sReceiveData,'L') <>0 THEN
				eErrorID:=MT_MCK_ERROR.FLT_PARA;//参数错误
				_diCmdState:=999;				
			END_IF
		END_IF

	3://清空发送与接收缓冲区
		_tonDelay(IN:= TRUE,pt:=T#1MS);//保证执行的是最新的一次
		SysMemSet( ADR( _Stemp ), 0, SIZEOF(_Stemp) );//清除缓存数据处理区域
		SysMemSet( ADR( _sSendData ), 0, SIZEOF(_sSendData) );//清除发送区域
		SysMemSet( ADR( _sReadDataTemp ), 0, SIZEOF(_sReadDataTemp) );//清除接收报告数据缓存区域
		SysMemSet( ADR( sFromServer ), 0, SIZEOF(sFromServer) );//清除发送区域
		_fbTcpIpClient.xNeedReceive := TRUE;//默认都是需要有收发交互的		
		IF _tonDelay.Q THEN
			_tonDelay(IN:= FALSE,pt:=T#20MS);
			_diCmdState:=_diCmdState+1;	
		END_IF
		
	4://拼接读取指令
		_tonDelay(IN:= _fbTcpIpClient.xRdyCmd ,pt:=T#1MS);
		_tonCmdTimeout(IN:= FALSE,pt:=T#2S);
		_sSendData := 'SI$R$N';//立即读取当前重量
		IF _tonDelay.Q THEN 
			_tonDelay(IN:= FALSE,pt:=T#20MS);
			_fbTcpIpClient.xEnable := FALSE;
			_diCmdState:=_diCmdState+1;		
		END_IF				
		
	5://发送指令,等待接收成功
		_tonCmdTimeout(IN:=TRUE ,pt:=T#2S);
		SysMemCpy(ADR(_fbTcpIpClient.aToServer),ADR(_sSendData),SIZEOF(_sSendData));	
		_fbTcpIpClient.udiSendNumber := LEN(_sSendData);				
		_fbTcpIpClient.xEnable := TRUE;	
		IF _fbTcpIpClient.xDone//接收成功
		THEN			
			_fbTcpIpClient.xEnable := FALSE;
			sFromServer := _sReceiveData := _fbTcpIpClient.sFromServer;//传递接收数据		
			rxBuffer := _fbTcpIpClient.rxBuffer;		
			IF FIND(_sReceiveData,'$R$N') <> 0 AND FIND(_sReceiveData,'S') <>0			
			THEN
				IF FIND(_sReceiveData,'mg') <> 0 THEN
					_Stemp[1]:=RIGHT(_sReceiveData,LEN(_sReceiveData)-5);
					_Stemp[2]:=LEFT(_Stemp[1],FIND(_Stemp[1],'mg$R$N')-1);
					stParOut.rCurrentWeight := TO_REAL(_Stemp[2]);
					stParOut.sWeightUnit:='mg';
				ELSE 
					IF FIND(_sReceiveData,'g') <> 0 THEN
						_Stemp[1]:=RIGHT(_sReceiveData,LEN(_sReceiveData)-5);
						_Stemp[2]:=LEFT(_Stemp[1],FIND(_Stemp[1],'g$R$N')-1);
						stParOut.rCurrentWeight := TO_REAL(_Stemp[2]);
						stParOut.sWeightUnit:='g';				
					END_IF				
				END_IF
				_diCmdState:=_diCmdState+1;
			ELSIF FIND(_sReceiveData,'EL') <>0 THEN
				eErrorID:=MT_MCK_ERROR.FLT_LogicaL;//逻辑错误
				_diCmdState:=999;
			ELSIF FIND(_sReceiveData,'ES') <>0 THEN
				eErrorID:=MT_MCK_ERROR.FLT_Syntax;//语法错误
				_diCmdState:=999;				
			ELSIF FIND(_sReceiveData,'I') <>0 THEN
				eErrorID:=MT_MCK_ERROR.FLT_CommandCantSend;//指令条件不满足,无法发送
				_diCmdState:=999;				
			ELSIF FIND(_sReceiveData,'L') <>0 THEN
				eErrorID:=MT_MCK_ERROR.FLT_PARA;//参数错误
				_diCmdState:=999;				
			END_IF
		END_IF
		IF _tonCmdTimeout.Q THEN
			eErrorID:=MT_MCK_ERROR.FLT_CMD_TIMEOUT;
			_diCmdState:=999;
		END_IF
	
	6://
		xComplete := TRUE; 
		
	ELSE
		;	
END_CASE
END_METHOD

METHOD PROTECTED CmdClearZero
VAR_OUTPUT
	xComplete: BOOL;
END_VAR
// return the real actual fault number
IF eERRORID <> MT_MCK_ERROR.No_ERROR
THEN
  RETURN;  
END_IF

CASE _diCmdState OF	
		
		
	0://清空发送与接收缓冲区
		_tonDelay(IN:= TRUE,pt:=T#1MS);//保证执行的是最新的一次
		_iNGCount:=0;
		SysMemSet( ADR( _sSendData ), 0, SIZEOF(_sSendData) );//清除发送区域
		SysMemSet( ADR( _sReadDataTemp ), 0, SIZEOF(_sReadDataTemp) );//清除接收报告数据缓存区域
		SysMemSet( ADR( sFromServer ), 0, SIZEOF(sFromServer) );//清除发送区域
		_fbTcpIpClient.xNeedReceive := TRUE;//默认都是需要有收发交互的		
		IF _tonDelay.Q THEN
			_tonDelay(IN:= FALSE,pt:=T#20MS);
			_diCmdState:=_diCmdState+1;	
		END_IF		
		
	1://拼接读取指令
		_tonDelay(IN:= _fbTcpIpClient.xRdyCmd ,pt:=T#2MS);
		_tonCmdTimeout(IN:= FALSE,pt:=T#2S);
		_sSendData := 'Z$R$N';//稳态清零
		IF _tonDelay.Q THEN 
			_tonDelay(IN:= FALSE,pt:=T#20MS);
			_fbTcpIpClient.xEnable := FALSE;
			_diCmdState:=_diCmdState+1;		
		END_IF		
		
	2://发送指令,等待接收成功
		_tonCmdTimeout(IN:=TRUE ,pt:=T#2S);
		SysMemCpy(ADR(_fbTcpIpClient.aToServer),ADR(_sSendData),SIZEOF(_sSendData));	
		_fbTcpIpClient.udiSendNumber := LEN(_sSendData);				
		_fbTcpIpClient.xEnable := TRUE;	
		IF _fbTcpIpClient.xDone//接收成功
		THEN			
			_tonCmdTimeout(IN:=FALSE ,pt:=T#2S);
			_fbTcpIpClient.xEnable := FALSE;
			sFromServer := _sReceiveData := _fbTcpIpClient.sFromServer;//传递接收数据		
			rxBuffer := _fbTcpIpClient.rxBuffer;		
			IF FIND(_sReceiveData,'$R$N') <> 0  						
			THEN
				IF FIND(_sReceiveData,'Z A') <> 0 THEN
					stParOut.rCurrentTareWight :=0;
					stParOut.rCurrentWeight :=0;
					_diCmdState:=_diCmdState+1;
				ELSE
					_iNGCount:=_iNGCount+1;
					IF _iNGCount< 3 THEN
						_diCmdState:=1;						
					ELSE
						IF FIND(_sReceiveData,'Z +') <> 0 THEN
							eErrorID:=MT_MCK_ERROR.FLT_ZOverMax;							
						ELSIF FIND(_sReceiveData,'Z -') <> 0 THEN
							eErrorID:=MT_MCK_ERROR.FLT_ZOverMin;				
						ELSIF FIND(_sReceiveData,'Z I') <> 0 THEN
							eErrorID:=MT_MCK_ERROR.FLT_ZI;					
						END_IF
						eErrorID:=MT_MCK_ERROR.FLT_CmdFeedback;//指令反馈出错
						_diCmdState:=999;
					END_IF
				END_IF
			END_IF
		END_IF
		IF _tonCmdTimeout.Q THEN
			eErrorID:=MT_MCK_ERROR.FLT_CMD_TIMEOUT;
			_diCmdState:=999;
		END_IF
	
	3://
		xComplete := TRUE; 
		
	ELSE
		;	
END_CASE
END_METHOD

METHOD PROTECTED CmdClearZeroInstanly
VAR_OUTPUT
	xComplete: BOOL;
END_VAR
// return the real actual fault number
IF eERRORID <> MT_MCK_ERROR.No_ERROR
THEN
  RETURN;  
END_IF

CASE _diCmdState OF	
		
		
	0://清空发送与接收缓冲区
		_tonDelay(IN:= TRUE,pt:=T#1MS);//保证执行的是最新的一次
		_iNGCount:=0;
		SysMemSet( ADR( _sSendData ), 0, SIZEOF(_sSendData) );//清除发送区域
		SysMemSet( ADR( _sReadDataTemp ), 0, SIZEOF(_sReadDataTemp) );//清除接收报告数据缓存区域
		SysMemSet( ADR( sFromServer ), 0, SIZEOF(sFromServer) );//清除发送区域
		_fbTcpIpClient.xNeedReceive := TRUE;//默认都是需要有收发交互的		
		IF _tonDelay.Q THEN
			_tonDelay(IN:= FALSE,pt:=T#20MS);
			_diCmdState:=_diCmdState+1;	
		END_IF		
		
	1://拼接读取指令
		_tonDelay(IN:= _fbTcpIpClient.xRdyCmd ,pt:=T#2MS);
		_tonCmdTimeout(IN:= FALSE,pt:=T#2S);
		_sSendData := 'ZI$R$N';//稳态清零
		IF _tonDelay.Q THEN 
			_tonDelay(IN:= FALSE,pt:=T#20MS);
			_fbTcpIpClient.xEnable := FALSE;
			_diCmdState:=_diCmdState+1;		
		END_IF		
		
	2://发送指令,等待接收成功
		_tonCmdTimeout(IN:=TRUE ,pt:=T#2S);
		SysMemCpy(ADR(_fbTcpIpClient.aToServer),ADR(_sSendData),SIZEOF(_sSendData));	
		_fbTcpIpClient.udiSendNumber := LEN(_sSendData);			
		_fbTcpIpClient.xEnable := TRUE;	
		IF _fbTcpIpClient.xDone//接收成功
		THEN			
			_tonCmdTimeout(IN:=FALSE ,pt:=T#2S);
			_fbTcpIpClient.xEnable := FALSE;
			sFromServer := _sReceiveData := _fbTcpIpClient.sFromServer;//传递接收数据		
			rxBuffer := _fbTcpIpClient.rxBuffer;		
			IF FIND(_sReceiveData,'$R$N') <> 0 						
			THEN
				IF FIND(_sReceiveData,'ZI') <> 0 AND (FIND(_sReceiveData,'S') <> 0 OR FIND(_sReceiveData,'D') <> 0) THEN
					stParOut.rCurrentTareWight :=0;
					stParOut.rCurrentWeight :=0;
					_diCmdState:=_diCmdState+1;
				ELSE
					_iNGCount:=_iNGCount+1;
					IF _iNGCount< 3 THEN
						_diCmdState:=1;						
					ELSE
						IF FIND(_sReceiveData,'Z +') <> 0 THEN
							eErrorID:=MT_MCK_ERROR.FLT_ZOverMax;							
						ELSIF FIND(_sReceiveData,'Z -') <> 0 THEN
							eErrorID:=MT_MCK_ERROR.FLT_ZOverMin;				
						ELSIF FIND(_sReceiveData,'Z I') <> 0 THEN
							eErrorID:=MT_MCK_ERROR.FLT_ZI;					
						END_IF
						eErrorID:=MT_MCK_ERROR.FLT_CmdFeedback;//指令反馈出错
						_diCmdState:=999;
					END_IF
				END_IF
			END_IF
		END_IF
		IF _tonCmdTimeout.Q THEN
			eErrorID:=MT_MCK_ERROR.FLT_CMD_TIMEOUT;
			_diCmdState:=999;
		END_IF
	
	3://
		xComplete := TRUE; 
		
	ELSE
		;	
END_CASE
END_METHOD

METHOD PROTECTED CmdCmd_AcquireWeight_Steady
VAR_OUTPUT
	xComplete: BOOL;
END_VAR
// return the real actual fault number
IF eERRORID <> MT_MCK_ERROR.No_ERROR
THEN
  RETURN;  
END_IF

CASE _diCmdState OF	
		
		
	0://清空发送与接收缓冲区
		_tonDelay(IN:= TRUE,pt:=T#1MS);//保证执行的是最新的一次
		SysMemSet( ADR( _Stemp ), 0, SIZEOF(_Stemp) );//清除缓存数据处理区域
		SysMemSet( ADR( _sSendData ), 0, SIZEOF(_sSendData) );//清除发送区域
		SysMemSet( ADR( _sReadDataTemp ), 0, SIZEOF(_sReadDataTemp) );//清除接收报告数据缓存区域
		SysMemSet( ADR( sFromServer ), 0, SIZEOF(sFromServer) );//清除发送区域
		_fbTcpIpClient.xNeedReceive := TRUE;//默认都是需要有收发交互的		
		IF _tonDelay.Q THEN
			_tonDelay(IN:= FALSE,pt:=T#20MS);
			_diCmdState:=_diCmdState+1;	
		END_IF		
		
	1://拼接读取指令
		_tonDelay(IN:= _fbTcpIpClient.xRdyCmd ,pt:=T#10MS);
		_tonCmdTimeout(IN:= FALSE,pt:=T#2S);
		_sSendData := 'S$R$N';
		IF _tonDelay.Q THEN 
			_tonDelay(IN:= FALSE,pt:=T#20MS);
			_fbTcpIpClient.xEnable := FALSE;
			_diCmdState:=_diCmdState+1;		
		END_IF		
		
	2://发送指令,等待接收成功
		_tonCmdTimeout(IN:=TRUE ,pt:=T#2S);
		SysMemCpy(ADR(_fbTcpIpClient.aToServer),ADR(_sSendData),SIZEOF(_sSendData));	
		_fbTcpIpClient.udiSendNumber := LEN(_sSendData);				
		_fbTcpIpClient.xEnable := TRUE;	
		IF _fbTcpIpClient.xDone//接收成功
		THEN			
			_fbTcpIpClient.xEnable := FALSE;
			sFromServer := _sReceiveData := _fbTcpIpClient.sFromServer;//传递接收数据		
			rxBuffer := _fbTcpIpClient.rxBuffer;		
			IF FIND(_sReceiveData,'$R$N') <> 0 AND FIND(_sReceiveData,'S') <>0			
			THEN
				IF FIND(_sReceiveData,'mg') <> 0 THEN
					_Stemp[1]:=RIGHT(_sReceiveData,LEN(_sReceiveData)-5);
					_Stemp[2]:=LEFT(_Stemp[1],FIND(_Stemp[1],'mg$R$N')-1);
					stParOut.rCurrentWeight := TO_REAL(_Stemp[2]);
					stParOut.sWeightUnit:='mg';
				ELSE 
					IF FIND(_sReceiveData,'g') <> 0 THEN
						_Stemp[1]:=RIGHT(_sReceiveData,LEN(_sReceiveData)-5);
						_Stemp[2]:=LEFT(_Stemp[1],FIND(_Stemp[1],'g$R$N')-1);
						stParOut.rCurrentWeight := TO_REAL(_Stemp[2]);
						stParOut.sWeightUnit:='g';				
					END_IF				
				END_IF
				_diCmdState:=_diCmdState+1;
			ELSIF FIND(_sReceiveData,'EL') <>0 THEN
				eErrorID:=MT_MCK_ERROR.FLT_LogicaL;//逻辑错误
				_diCmdState:=999;
			ELSIF FIND(_sReceiveData,'ES') <>0 THEN
				eErrorID:=MT_MCK_ERROR.FLT_Syntax;//语法错误
				_diCmdState:=999;				
			ELSIF FIND(_sReceiveData,'I') <>0 THEN
				eErrorID:=MT_MCK_ERROR.FLT_CommandCantSend;//指令条件不满足,无法发送
				_diCmdState:=999;				
			ELSIF FIND(_sReceiveData,'L') <>0 THEN
				eErrorID:=MT_MCK_ERROR.FLT_PARA;//参数错误
				_diCmdState:=999;				
			END_IF
		END_IF
		IF _tonCmdTimeout.Q THEN
			eErrorID:=MT_MCK_ERROR.FLT_CMD_TIMEOUT;
			_diCmdState:=999;
		END_IF
	
	3://
		xComplete := TRUE; 
		
	ELSE
		;	
END_CASE
END_METHOD

METHOD PROTECTED CmdRestart
VAR_OUTPUT
	xComplete: BOOL;
END_VAR
// return the real actual fault number
IF eERRORID <> MT_MCK_ERROR.No_ERROR
THEN
  RETURN;  
END_IF

CASE _diCmdState OF	
		
		
	0://清空发送与接收缓冲区
		xRefOk:=FALSE;
		_tonDelay(IN:= TRUE,pt:=T#20MS);//保证执行的是最新的一次
		SysMemSet( ADR( _sSendData ), 0, SIZEOF(_sSendData) );//清除发送区域
		SysMemSet( ADR( _sReadDataTemp ), 0, SIZEOF(_sReadDataTemp) );//清除接收报告数据缓存区域
		SysMemSet( ADR( sFromServer ), 0, SIZEOF(sFromServer) );//清除发送区域
		_fbTcpIpClient.xNeedReceive := TRUE;//默认都是需要有收发交互的		
		IF _tonDelay.Q THEN
			_tonDelay(IN:= FALSE,pt:=T#20MS);
			_diCmdState:=_diCmdState+1;	
		END_IF		
		
	1://拼接读取指令
		_tonDelay(IN:= _fbTcpIpClient.xRdyCmd ,pt:=T#10MS);
		_tonCmdTimeout(IN:= FALSE,pt:=T#2S);
		_sSendData := 'R01$R$N';
		IF _tonDelay.Q THEN 
			_tonDelay(IN:= FALSE,pt:=T#20MS);
			_fbTcpIpClient.xEnable := FALSE;
			_diCmdState:=_diCmdState+1;		
		END_IF		
		
	2://发送指令,等待接收成功
		_tonCmdTimeout(IN:=TRUE ,pt:=T#6S);
		SysMemCpy(ADR(_fbTcpIpClient.aToServer),ADR(_sSendData),SIZEOF(_sSendData));	
		_fbTcpIpClient.udiSendNumber := LEN(_sSendData);				
		_fbTcpIpClient.xEnable := TRUE;	
		IF _fbTcpIpClient.xDone//接收成功
		THEN			
			_fbTcpIpClient.xEnable := FALSE;
			sFromServer := _sReceiveData := _fbTcpIpClient.sFromServer;//传递接收数据		
			rxBuffer := _fbTcpIpClient.rxBuffer;		
			IF FIND(_sReceiveData,'$R$N') <> 0 AND FIND(_sReceiveData,'I4') <> 0						
			THEN
				CutStrToSeperator('"',_sReceiveData);
				stParOut.sSrialNumber := CutStrToSeperator('"',_sReceiveData);
				_diCmdState:=_diCmdState+1;	
			END_IF
		END_IF
		IF _tonCmdTimeout.Q THEN
			eErrorID:=MT_MCK_ERROR.FLT_CMD_TIMEOUT;
			_diCmdState:=999;
		END_IF
		
		
	3://
		xRefOk:=TRUE;
		xComplete := TRUE; 
		
	ELSE
		;	
END_CASE
END_METHOD

METHOD PROTECTED CmdSerialNum
VAR_OUTPUT
	xComplete: BOOL;
END_VAR
// return the real actual fault number
IF eERRORID <> MT_MCK_ERROR.No_ERROR
THEN
  RETURN;  
END_IF

CASE _diCmdState OF	
		
		
	0://清空发送与接收缓冲区
		xRefOk:=FALSE;
		_tonDelay(IN:= TRUE,pt:=T#20MS);//保证执行的是最新的一次
		SysMemSet( ADR( _sSendData ), 0, SIZEOF(_sSendData) );//清除发送区域
		SysMemSet( ADR( _sReadDataTemp ), 0, SIZEOF(_sReadDataTemp) );//清除接收报告数据缓存区域
		SysMemSet( ADR( sFromServer ), 0, SIZEOF(sFromServer) );//清除发送区域
		_fbTcpIpClient.xNeedReceive := TRUE;//默认都是需要有收发交互的		
		IF _tonDelay.Q THEN
			_tonDelay(IN:= FALSE,pt:=T#20MS);
			_diCmdState:=_diCmdState+1;	
		END_IF		
		
	1://拼接读取指令
		_tonDelay(IN:= _fbTcpIpClient.xRdyCmd ,pt:=T#10MS);
		_tonCmdTimeout(IN:= FALSE,pt:=T#2S);
		_sSendData := 'I4$R$N';
		IF _tonDelay.Q THEN 
			_tonDelay(IN:= FALSE,pt:=T#20MS);
			_fbTcpIpClient.xEnable := FALSE;
			_diCmdState:=_diCmdState+1;		
		END_IF		
		
	2://发送指令,等待接收成功
		SysMemCpy(ADR(_fbTcpIpClient.aToServer),ADR(_sSendData),SIZEOF(_sSendData));	
		_fbTcpIpClient.udiSendNumber := LEN(_sSendData);				
		_fbTcpIpClient.xEnable := TRUE;	
		IF _fbTcpIpClient.xDone//接收成功
		THEN			
			_fbTcpIpClient.xEnable := FALSE;
			sFromServer := _sReceiveData := _fbTcpIpClient.sFromServer;//传递接收数据		
			rxBuffer := _fbTcpIpClient.rxBuffer;		
			IF FIND(_sReceiveData,'$R$N') <> 0 AND FIND(_sReceiveData,'I4') <> 0						
			THEN
				CutStrToSeperator('"',_sReceiveData);
				stParOut.sSrialNumber := CutStrToSeperator('"',_sReceiveData);
				_diCmdState:=_diCmdState+1;	
		  ELSE
				_diCmdState:=_diCmdState+1;	
			END_IF
		 END_IF
		IF _fbTcpIpClient.xError 
		THEN//以太网功能报警，一般就是网络建立有问题，此时一般需要去查网络问题
			IF _iSendNgCount < 2//3次重发
			THEN		
				_tDelay(in:=TRUE,PT:=T#100MS);	
				IF _tDelay.Q
				THEN
			    _iSendNgCount := _iSendNgCount + 1;					
					_tDelay(in:=FALSE);
					_diCmdState:=1;//重发
				END_IF							
			ELSE						
					eErrorID:=MT_MCK_ERROR.FLT_CommandCantSend;
					_diCmdState := 999;
			END_IF						
		END_IF 
	
	3://
		xRefOk:=TRUE;
		xComplete := TRUE; 
		
	ELSE
		;	
END_CASE
END_METHOD

METHOD PROTECTED CmdSetTare
VAR_OUTPUT
	xComplete: BOOL;
END_VAR
// return the real actual fault number
IF eERRORID <> MT_MCK_ERROR.No_ERROR
THEN
  RETURN;  
END_IF

CASE _diCmdState OF	
	0://清空发送与接收缓冲区
		_tonDelay(IN:= TRUE,pt:=T#20MS);//保证执行的是最新的一次
		SysMemSet( ADR( _Stemp ), 0, SIZEOF(_Stemp) );//清除缓存数据处理区域
		SysMemSet( ADR( _sSendData ), 0, SIZEOF(_sSendData) );//清除发送区域
		SysMemSet( ADR( _sReadDataTemp ), 0, SIZEOF(_sReadDataTemp) );//清除接收报告数据缓存区域
		SysMemSet( ADR( sFromServer ), 0, SIZEOF(sFromServer) );//清除发送区域
		_fbTcpIpClient.xNeedReceive := TRUE;//默认都是需要有收发交互的		
		IF _tonDelay.Q THEN
			_tonDelay(IN:= FALSE,pt:=T#20MS);
			_diCmdState:=_diCmdState+1;	
		END_IF			
		
	1://拼接读取指令
		_tonDelay(IN:= _fbTcpIpClient.xRdyCmd ,pt:=T#10MS);
		_tonCmdTimeout(IN:= FALSE,pt:=T#2S);
		_sSendData := CONCAT(_sSendData,'TA');
		_sSendData := CONCAT(_sSendData,' ');		
		_sSendData := CONCAT(_sSendData,TO_STRING(rTareSet));
		_sSendData := CONCAT(_sSendData,' ');
		_sSendData := CONCAT(_sSendData,'g');//单位
		_sSendData := CONCAT(_sSendData,'$R$N');//回车换行符				
		IF _tonDelay.Q THEN 
			_tonDelay(IN:= FALSE,pt:=T#20MS);
			_fbTcpIpClient.xEnable := FALSE;
			_diCmdState:=_diCmdState+1;		
		END_IF
	
	2://发送指令,等待接收成功
		_tonCmdTimeout(IN:=TRUE ,pt:=T#2S);
		SysMemCpy(ADR(_fbTcpIpClient.aToServer),ADR(_sSendData),SIZEOF(_sSendData));	
		_fbTcpIpClient.udiSendNumber := LEN(_sSendData);				
		_fbTcpIpClient.xEnable := TRUE;	
		IF _fbTcpIpClient.xDone//接收成功
		THEN			
			_fbTcpIpClient.xEnable := FALSE;
			sFromServer := _sReceiveData := _fbTcpIpClient.sFromServer;//传递接收数据		
			rxBuffer := _fbTcpIpClient.rxBuffer;		
			IF FIND(_sReceiveData,'$R$N') <> 0 AND FIND(_sReceiveData,'TA') <> 0						
			THEN
				_Stemp[1]:=RIGHT(_sReceiveData,LEN(_sReceiveData)-5);
				_Stemp[2]:=LEFT(_Stemp[1],FIND(_Stemp[1],'g$R$N')-1);
				stParOut.rCurrentTareWight := TO_REAL(_Stemp[2]);
				_diCmdState:=_diCmdState+1;	
			END_IF
		END_IF		
		IF _tonCmdTimeout.Q THEN
			eErrorID:=MT_MCK_ERROR.FLT_CMD_TIMEOUT;
			_diCmdState:=999;
		END_IF
		
	3://清空发送与接收缓冲区
		_tonDelay(IN:= TRUE,pt:=T#20MS);//保证执行的是最新的一次
		SysMemSet( ADR( _Stemp ), 0, SIZEOF(_Stemp) );//清除缓存数据处理区域
		SysMemSet( ADR( _sSendData ), 0, SIZEOF(_sSendData) );//清除发送区域
		SysMemSet( ADR( _sReadDataTemp ), 0, SIZEOF(_sReadDataTemp) );//清除接收报告数据缓存区域
		SysMemSet( ADR( sFromServer ), 0, SIZEOF(sFromServer) );//清除发送区域
		_fbTcpIpClient.xNeedReceive := TRUE;//默认都是需要有收发交互的		
		IF _tonDelay.Q THEN
			_tonDelay(IN:= FALSE,pt:=T#20MS);
			_diCmdState:=_diCmdState+1;	
		END_IF		

	4://拼接读取指令
		_tonDelay(IN:= _fbTcpIpClient.xRdyCmd ,pt:=T#10MS);
		_tonCmdTimeout(IN:= FALSE,pt:=T#2S);
		_sSendData := 'SI$R$N';
		IF _tonDelay.Q THEN 
			_tonDelay(IN:= FALSE,pt:=T#20MS);
			_fbTcpIpClient.xEnable := FALSE;
			_diCmdState:=_diCmdState+1;		
		END_IF		
		
	5://发送指令,等待接收成功
		_tonCmdTimeout(IN:=TRUE ,pt:=T#2S);
		SysMemCpy(ADR(_fbTcpIpClient.aToServer),ADR(_sSendData),SIZEOF(_sSendData));	
		_fbTcpIpClient.udiSendNumber := LEN(_sSendData);				
		_fbTcpIpClient.xEnable := TRUE;	
		IF _fbTcpIpClient.xDone//接收成功
		THEN			
			_fbTcpIpClient.xEnable := FALSE;
			sFromServer := _sReceiveData := _fbTcpIpClient.sFromServer;//传递接收数据		
			rxBuffer := _fbTcpIpClient.rxBuffer;		
			IF FIND(_sReceiveData,'$R$N') <> 0 AND FIND(_sReceiveData,'S') <>0			
			THEN
				IF FIND(_sReceiveData,'mg') <> 0 THEN
					_Stemp[1]:=RIGHT(_sReceiveData,LEN(_sReceiveData)-5);
					_Stemp[2]:=LEFT(_Stemp[1],FIND(_Stemp[1],'mg$R$N')-1);
					stParOut.rCurrentWeight := TO_REAL(_Stemp[2]);
					stParOut.sWeightUnit:='mg';
				ELSE 
					IF FIND(_sReceiveData,'g') <> 0 THEN
						_Stemp[1]:=RIGHT(_sReceiveData,LEN(_sReceiveData)-5);
						_Stemp[2]:=LEFT(_Stemp[1],FIND(_Stemp[1],'g$R$N')-1);
						stParOut.rCurrentWeight := TO_REAL(_Stemp[2]);
						stParOut.sWeightUnit:='g';				
					END_IF				
				END_IF
				_diCmdState:=_diCmdState+1;
			ELSIF FIND(_sReceiveData,'EL') <>0 THEN
				eErrorID:=MT_MCK_ERROR.FLT_LogicaL;//逻辑错误
				_diCmdState:=999;
			ELSIF FIND(_sReceiveData,'ES') <>0 THEN
				eErrorID:=MT_MCK_ERROR.FLT_Syntax;//语法错误
				_diCmdState:=999;				
			ELSIF FIND(_sReceiveData,'I') <>0 THEN
				eErrorID:=MT_MCK_ERROR.FLT_CommandCantSend;//指令条件不满足,无法发送
				_diCmdState:=999;				
			ELSIF FIND(_sReceiveData,'L') <>0 THEN
				eErrorID:=MT_MCK_ERROR.FLT_PARA;//参数错误
				_diCmdState:=999;				
			END_IF			
		END_IF
		IF _tonCmdTimeout.Q THEN
			eErrorID:=MT_MCK_ERROR.FLT_CMD_TIMEOUT;
			_diCmdState:=999;
		END_IF		
		
	6://
		xComplete := TRUE; 
		
	ELSE
		;	
END_CASE
END_METHOD

METHOD PROTECTED CmdShelling
VAR_OUTPUT
	xComplete: BOOL;
END_VAR
// return the real actual fault number
IF eERRORID <> MT_MCK_ERROR.No_ERROR
THEN
  RETURN;  
END_IF

CASE _diCmdState OF	
	0://清空发送与接收缓冲区
		_tonDelay(IN:= TRUE,pt:=T#20MS);//保证执行的是最新的一次
		SysMemSet( ADR( _Stemp ), 0, SIZEOF(_Stemp) );//清除缓存数据处理区域
		SysMemSet( ADR( _sSendData ), 0, SIZEOF(_sSendData) );//清除发送区域
		SysMemSet( ADR( _sReadDataTemp ), 0, SIZEOF(_sReadDataTemp) );//清除接收报告数据缓存区域
		SysMemSet( ADR( sFromServer ), 0, SIZEOF(sFromServer) );//清除发送区域
		_fbTcpIpClient.xNeedReceive := TRUE;//默认都是需要有收发交互的		
		IF _tonDelay.Q THEN
			_tonDelay(IN:= FALSE,pt:=T#20MS);
			_diCmdState:=_diCmdState+1;	
		END_IF		
		
	1://拼接读取指令
		_tonDelay(IN:= _fbTcpIpClient.xRdyCmd ,pt:=T#10MS);
		_tonCmdTimeout(IN:= FALSE,pt:=T#2S);
		_sSendData := 'T$R$N';//稳态去皮重
		IF _tonDelay.Q THEN 
			_tonDelay(IN:= FALSE,pt:=T#20MS);
			_fbTcpIpClient.xEnable := FALSE;
			_diCmdState:=_diCmdState+1;		
		END_IF		
		
	2://发送指令,等待接收成功
		_tonCmdTimeout(IN:=TRUE ,pt:=T#2S);
		SysMemCpy(ADR(_fbTcpIpClient.aToServer),ADR(_sSendData),SIZEOF(_sSendData));	
		_fbTcpIpClient.udiSendNumber := LEN(_sSendData);				
		_fbTcpIpClient.xEnable := TRUE;	
		IF _fbTcpIpClient.xDone//接收成功
		THEN			
			_fbTcpIpClient.xEnable := FALSE;
			sFromServer := _sReceiveData := _fbTcpIpClient.sFromServer;//传递接收数据		
			rxBuffer := _fbTcpIpClient.rxBuffer;		
			IF FIND(_sReceiveData,'$R$N') <> 0 						
			THEN
				IF FIND(_sReceiveData,'S') <> 0 THEN
					_Stemp[1]:=RIGHT(_sReceiveData,LEN(_sReceiveData)-4);
					_Stemp[2]:=LEFT(_Stemp[1],FIND(_Stemp[1],'g$R$N')-1);
					stParOut.rCurrentTareWight := TO_REAL(_Stemp[2]);
					_diCmdState:=_diCmdState+1;
				ELSIF FIND(_sReceiveData,'T +') <> 0 THEN	
					eErrorID:=MT_MCK_ERROR.FLT_ZOverMax;
					_diCmdState:=999;
				ELSIF FIND(_sReceiveData,'T -') <> 0 THEN	
					eErrorID:=MT_MCK_ERROR.FLT_ZOverMax;
					_diCmdState:=999;
				END_IF										
			END_IF
		END_IF		
		IF _tonCmdTimeout.Q THEN
			eErrorID:=MT_MCK_ERROR.FLT_CMD_TIMEOUT;
			_diCmdState:=999;
		END_IF
		
	3://清空发送与接收缓冲区
		_tonDelay(IN:= TRUE,pt:=T#20MS);//保证执行的是最新的一次
		SysMemSet( ADR( _Stemp ), 0, SIZEOF(_Stemp) );//清除缓存数据处理区域
		SysMemSet( ADR( _sSendData ), 0, SIZEOF(_sSendData) );//清除发送区域
		SysMemSet( ADR( _sReadDataTemp ), 0, SIZEOF(_sReadDataTemp) );//清除接收报告数据缓存区域
		SysMemSet( ADR( sFromServer ), 0, SIZEOF(sFromServer) );//清除发送区域
		_fbTcpIpClient.xNeedReceive := TRUE;//默认都是需要有收发交互的		
		IF _tonDelay.Q THEN
			_tonDelay(IN:= FALSE,pt:=T#20MS);
			_diCmdState:=_diCmdState+1;	
		END_IF		

	4://拼接读取指令
		_tonDelay(IN:= _fbTcpIpClient.xRdyCmd ,pt:=T#10MS);
		_tonCmdTimeout(IN:= FALSE,pt:=T#2S);
		_sSendData := 'SI$R$N';
		IF _tonDelay.Q THEN 
			_tonDelay(IN:= FALSE,pt:=T#20MS);
			_fbTcpIpClient.xEnable := FALSE;
			_diCmdState:=_diCmdState+1;		
		END_IF		
		
	5://发送指令,等待接收成功
		_tonCmdTimeout(IN:=TRUE ,pt:=T#2S);
		SysMemCpy(ADR(_fbTcpIpClient.aToServer),ADR(_sSendData),SIZEOF(_sSendData));	
		_fbTcpIpClient.udiSendNumber := LEN(_sSendData);				
		_fbTcpIpClient.xEnable := TRUE;	
		IF _fbTcpIpClient.xDone//接收成功
		THEN			
			_fbTcpIpClient.xEnable := FALSE;
			sFromServer := _sReceiveData := _fbTcpIpClient.sFromServer;//传递接收数据		
			rxBuffer := _fbTcpIpClient.rxBuffer;		
			IF FIND(_sReceiveData,'$R$N') <> 0 AND FIND(_sReceiveData,'S') <>0			
			THEN
				IF FIND(_sReceiveData,'mg') <> 0 THEN
					_Stemp[1]:=RIGHT(_sReceiveData,LEN(_sReceiveData)-5);
					_Stemp[2]:=LEFT(_Stemp[1],FIND(_Stemp[1],'mg$R$N')-1);
					stParOut.rCurrentWeight := TO_REAL(_Stemp[2]);
					stParOut.sWeightUnit:='mg';
				ELSE 
					IF FIND(_sReceiveData,'g') <> 0 THEN
						_Stemp[1]:=RIGHT(_sReceiveData,LEN(_sReceiveData)-5);
						_Stemp[2]:=LEFT(_Stemp[1],FIND(_Stemp[1],'g$R$N')-1);
						stParOut.rCurrentWeight := TO_REAL(_Stemp[2]);
						stParOut.sWeightUnit:='g';				
					END_IF				
				END_IF
				_diCmdState:=_diCmdState+1;
			ELSIF FIND(_sReceiveData,'EL') <>0 THEN
				eErrorID:=MT_MCK_ERROR.FLT_LogicaL;//逻辑错误
				_diCmdState:=999;
			ELSIF FIND(_sReceiveData,'ES') <>0 THEN
				eErrorID:=MT_MCK_ERROR.FLT_Syntax;//语法错误
				_diCmdState:=999;				
			ELSIF FIND(_sReceiveData,'I') <>0 THEN
				eErrorID:=MT_MCK_ERROR.FLT_CommandCantSend;//指令条件不满足,无法发送
				_diCmdState:=999;				
			ELSIF FIND(_sReceiveData,'L') <>0 THEN
				eErrorID:=MT_MCK_ERROR.FLT_PARA;//参数错误
				_diCmdState:=999;				
			END_IF			
		END_IF
		IF _tonCmdTimeout.Q THEN
			eErrorID:=MT_MCK_ERROR.FLT_CMD_TIMEOUT;
			_diCmdState:=999;
		END_IF

	
	6://
		xComplete := TRUE; 
		
	ELSE
		;	
END_CASE
END_METHOD

METHOD PROTECTED CmdShellingInstanly
VAR_OUTPUT
	xComplete: BOOL;
END_VAR
// return the real actual fault number
IF eERRORID <> MT_MCK_ERROR.No_ERROR
THEN
  RETURN;  
END_IF

CASE _diCmdState OF	
	0://清空发送与接收缓冲区
		_tonDelay(IN:= TRUE,pt:=T#20MS);//保证执行的是最新的一次
		SysMemSet( ADR( _Stemp ), 0, SIZEOF(_Stemp) );//清除缓存数据处理区域
		SysMemSet( ADR( _sSendData ), 0, SIZEOF(_sSendData) );//清除发送区域
		SysMemSet( ADR( _sReadDataTemp ), 0, SIZEOF(_sReadDataTemp) );//清除接收报告数据缓存区域
		SysMemSet( ADR( sFromServer ), 0, SIZEOF(sFromServer) );//清除发送区域
		_fbTcpIpClient.xNeedReceive := TRUE;//默认都是需要有收发交互的		
		IF _tonDelay.Q THEN
			_tonDelay(IN:= FALSE,pt:=T#20MS);
			_diCmdState:=_diCmdState+1;	
		END_IF		
		
	1://拼接读取指令
		_tonDelay(IN:= _fbTcpIpClient.xRdyCmd ,pt:=T#10MS);
		_tonCmdTimeout(IN:= FALSE,pt:=T#2S);
		_sSendData := 'TI$R$N';//立即去皮重
		IF _tonDelay.Q THEN 
			_tonDelay(IN:= FALSE,pt:=T#20MS);
			_fbTcpIpClient.xEnable := FALSE;
			_diCmdState:=_diCmdState+1;		
		END_IF		
		
	2://发送指令,等待接收成功
		_tonCmdTimeout(IN:=TRUE ,pt:=T#2S);
		SysMemCpy(ADR(_fbTcpIpClient.aToServer),ADR(_sSendData),SIZEOF(_sSendData));	
		_fbTcpIpClient.udiSendNumber := LEN(_sSendData);			
		_fbTcpIpClient.xEnable := TRUE;	
		IF _fbTcpIpClient.xDone//接收成功
		THEN			
			_fbTcpIpClient.xEnable := FALSE;
			sFromServer := _sReceiveData := _fbTcpIpClient.sFromServer;//传递接收数据		
			rxBuffer := _fbTcpIpClient.rxBuffer;		
			IF FIND(_sReceiveData,'$R$N') <> 0 						
			THEN
				IF FIND(_sReceiveData,'TI S') <> 0 OR FIND(_sReceiveData,'TI D') <> 0 THEN
					_Stemp[1]:=RIGHT(_sReceiveData,LEN(_sReceiveData)-4);
					_Stemp[2]:=LEFT(_Stemp[1],FIND(_Stemp[1],'g$R$N')-1);
					stParOut.rCurrentTareWight := TO_REAL(_Stemp[2]);
					_diCmdState:=_diCmdState+1;
				ELSIF FIND(_sReceiveData,'TI +') <> 0 THEN	
					eErrorID:=MT_MCK_ERROR.FLT_ZOverMax;
					_diCmdState:=999;
				ELSIF FIND(_sReceiveData,'TI -') <> 0 THEN	
					eErrorID:=MT_MCK_ERROR.FLT_ZOverMax;
					_diCmdState:=999;
				END_IF										
			END_IF
		END_IF		
		IF _tonCmdTimeout.Q THEN
			eErrorID:=MT_MCK_ERROR.FLT_CMD_TIMEOUT;
			_diCmdState:=999;
		END_IF
		
	3://清空发送与接收缓冲区
		_tonDelay(IN:= TRUE,pt:=T#20MS);//保证执行的是最新的一次
		SysMemSet( ADR( _Stemp ), 0, SIZEOF(_Stemp) );//清除缓存数据处理区域
		SysMemSet( ADR( _sSendData ), 0, SIZEOF(_sSendData) );//清除发送区域
		SysMemSet( ADR( _sReadDataTemp ), 0, SIZEOF(_sReadDataTemp) );//清除接收报告数据缓存区域
		SysMemSet( ADR( sFromServer ), 0, SIZEOF(sFromServer) );//清除发送区域
		_fbTcpIpClient.xNeedReceive := TRUE;//默认都是需要有收发交互的		
		IF _tonDelay.Q THEN
			_tonDelay(IN:= FALSE,pt:=T#20MS);
			_diCmdState:=_diCmdState+1;	
		END_IF		

	4://拼接读取指令
		_tonDelay(IN:= _fbTcpIpClient.xRdyCmd ,pt:=T#10MS);
		_tonCmdTimeout(IN:= FALSE,pt:=T#2S);
		_sSendData := 'SI$R$N';
		IF _tonDelay.Q THEN 
			_tonDelay(IN:= FALSE,pt:=T#20MS);
			_fbTcpIpClient.xEnable := FALSE;
			_diCmdState:=_diCmdState+1;		
		END_IF		
		
	5://发送指令,等待接收成功
		_tonCmdTimeout(IN:=TRUE ,pt:=T#2S);
		SysMemCpy(ADR(_fbTcpIpClient.aToServer),ADR(_sSendData),SIZEOF(_sSendData));	
		_fbTcpIpClient.udiSendNumber := LEN(_sSendData);				
		_fbTcpIpClient.xEnable := TRUE;	
		IF _fbTcpIpClient.xDone//接收成功
		THEN			
			_fbTcpIpClient.xEnable := FALSE;
			sFromServer := _sReceiveData := _fbTcpIpClient.sFromServer;//传递接收数据		
			rxBuffer := _fbTcpIpClient.rxBuffer;		
			IF FIND(_sReceiveData,'$R$N') <> 0 AND FIND(_sReceiveData,'S') <>0			
			THEN
				IF FIND(_sReceiveData,'mg') <> 0 THEN
					_Stemp[1]:=RIGHT(_sReceiveData,LEN(_sReceiveData)-5);
					_Stemp[2]:=LEFT(_Stemp[1],FIND(_Stemp[1],'mg$R$N')-1);
					stParOut.rCurrentWeight := TO_REAL(_Stemp[2]);
					stParOut.sWeightUnit:='mg';
				ELSE 
					IF FIND(_sReceiveData,'g') <> 0 THEN
						_Stemp[1]:=RIGHT(_sReceiveData,LEN(_sReceiveData)-5);
						_Stemp[2]:=LEFT(_Stemp[1],FIND(_Stemp[1],'g$R$N')-1);
						stParOut.rCurrentWeight := TO_REAL(_Stemp[2]);
						stParOut.sWeightUnit:='g';				
					END_IF				
				END_IF
				_diCmdState:=_diCmdState+1;
			ELSIF FIND(_sReceiveData,'EL') <>0 THEN
				eErrorID:=MT_MCK_ERROR.FLT_LogicaL;//逻辑错误
				_diCmdState:=999;
			ELSIF FIND(_sReceiveData,'ES') <>0 THEN
				eErrorID:=MT_MCK_ERROR.FLT_Syntax;//语法错误
				_diCmdState:=999;				
			ELSIF FIND(_sReceiveData,'I') <>0 THEN
				eErrorID:=MT_MCK_ERROR.FLT_CommandCantSend;//指令条件不满足,无法发送
				_diCmdState:=999;				
			ELSIF FIND(_sReceiveData,'L') <>0 THEN
				eErrorID:=MT_MCK_ERROR.FLT_PARA;//参数错误
				_diCmdState:=999;				
			END_IF			
		END_IF
		IF _tonCmdTimeout.Q THEN
			eErrorID:=MT_MCK_ERROR.FLT_CMD_TIMEOUT;
			_diCmdState:=999;
		END_IF

	
	6://
		xComplete := TRUE; 
		
	ELSE
		;	
END_CASE
END_METHOD

{attribute 'tc_no_symbol'}
METHOD PROTECTED CyclicAction
VAR_INPUT
END_VAR
VAR_OUTPUT
	xComplete: BOOL;
END_VAR
VAR	
END_VAR
IF xAbort=0 THEN
	IF xFirstInvocation THEN//执行初始化
	(*
	* Staring
	* for then first (!) invocaion,
	* sample then input variables
	*)
		SysMemSet(ADR(_sReceiveData),0,SIZEOF(_sReceiveData));//清空接收数据
		SysMemSet(ADR(sFromServer),0,SIZEOF(sFromServer));//清空数据
		//_iSendNgCount := _iReadNGCount := _iReadDataCount := 0;//控制重发次数
		xFirstInvocation:=0;
	END_IF   

//检测停止指令是否发生
_rStopCmdTrig(CLK:= NOT xEStop OR (stDeviceOpe.xAcquireWeight_Stop_HMI AND NOT xAutoMode AND NOT xDeviceRunning) OR (stDeviceOpe.xAcquireWeight_Stop_Auto AND (xAutoMode OR xDeviceRunning)));	
IF _rStopCmdTrig.Q//检测到停止指令
THEN
	_diCmdState := 0;
	eCmd := MT_MCK_CMD.Cmd_AcquireWeight_Stop;
	_tonCmdTimeout(in:=FALSE);
	_tonDelay(IN:= FALSE);
	_tonTimeout(in:=FALSE);
END_IF

	REPEAT 	
			IF	stSysPar.sRemoteHost = ''  OR //检测参数是否配置正确		
				stSysPar.nRemotePort = 0			 				 	 
			THEN
				eERRORID := MT_MCK_ERROR.FLT_PARA;//参数配置错误
			END_IF	

			CASE eCmd OF//判断指令类型
				MT_MCK_CMD.Cmd_SerialNum://获取序列号
					CmdSerialNum(xComplete=> xComplete);
					
				MT_MCK_CMD.Cmd_AcquireWeight_RealTime://获取及时重量
					CmdAcquireWeight_RealTime(xComplete=> xComplete);

				MT_MCK_CMD.Cmd_AcquireWeight_Steady://获取稳态重量
					CmdCmd_AcquireWeight_Steady(xComplete=> xComplete);

				MT_MCK_CMD.Cmd_AcquireWeight_Continuous://获取连续重量
					CmdAcquireWeight_Continuous(xComplete=> xComplete);
					
				MT_MCK_CMD.Cmd_AcquireWeight_Stop://停止获取重量
					CmdAcquireWeight_Stop(xComplete=> xComplete);	

				MT_MCK_CMD.Cmd_ShellingInstanly://立即去皮
					CmdShellingInstanly(xComplete=> xComplete);

				MT_MCK_CMD.Cmd_Shelling://稳态去皮
					CmdShelling(xComplete=> xComplete);	

				MT_MCK_CMD.Cmd_SetTare://设置皮重
					CmdSetTare(xComplete=> xComplete);

				MT_MCK_CMD.Cmd_ClearTare://清除皮重
					CmdClearTare(xComplete=> xComplete);	

				MT_MCK_CMD.Cmd_ClearZero://稳态清零
					CmdClearZero(xComplete=> xComplete);
					
				MT_MCK_CMD.Cmd_ClearZeroInstanly://立即清零
					CmdClearZeroInstanly(xComplete=> xComplete);	

				MT_MCK_CMD.Cmd_Restart://重启
					CmdRestart(xComplete=> xComplete);				
			ELSE
				;	
			END_CASE
	   
		UNTIL (TRUE)//处于一直刷新阶段
	END_REPEAT
END_IF

IF NOT xExecute OR xComplete OR eErrorID<>MT_MCK_ERROR.No_ERROR THEN    
    (*
    * Cleaning
    * => free as much allocated resources as possible
    *)    
    tOperationTimer(IN:=0);
END_IF
END_METHOD

{attribute 'tc_no_symbol'}
METHOD PRIVATE FINAL HandleAbortedSTATE
VAR_INPUT
END_VAR
VAR_OUTPUT
	xAgain: BOOL;
END_VAR
VAR
{attribute 'tc_no_symbol'}	
	xComplete: BOOL;
END_VAR
IF xAborted AND xResetRequest THEN
    eState:=STATE.RESETING;
    xAgain:=1;
ELSE
    xBusy:=0;
    xAborted:=1;
    //xResetRequest:=(xExecute=0);
    xAgain:=0;(* !!! *)
END_IF
END_METHOD

{attribute 'tc_no_symbol'}
METHOD PRIVATE FINAL HandleAbortingSTATE
VAR_INPUT
END_VAR
VAR_OUTPUT
	xAgain: BOOL;
END_VAR
VAR
{attribute 'tc_no_symbol'}	
	xComplete: BOOL;
END_VAR
AbortAction(xComplete=> xComplete, eErrorID=> eErrorID);

IF eErrorID<>MT_MCK_ERROR.NO_ERROR THEN
    eState:=STATE.INERROR;
    xAgain:=1;
ELSIF xComplete THEN
    eState:=STATE.ABORTED;
    xAgain:=1;
END_IF
END_METHOD

{attribute 'tc_no_symbol'}
METHOD PRIVATE FINAL HandleDoneSTATE
VAR_INPUT
END_VAR
VAR_OUTPUT
	xAgain: BOOL;
END_VAR
//在运行过程中要是切换模式，再运行完成之后，检测到模式的切换，就需要回到初始位置，进行下一次执行准备
IF _xDone AND ((xExecute=0) OR ( _xModeChange AND NOT _xAutoOpe)  OR ( NOT xAutoMode AND NOT xDeviceRunning AND ( NOT _xAutoOpe OR _xHMIOpe))) THEN
	eState:=STATE.RESETING;
	xAgain:=1;
ELSE
	xBusy:=0;
	_xDone:=1;
	//xResetRequest:=(xExecute=0);
	xAgain:=0;(* !!! *)
END_IF
END_METHOD

{attribute 'tc_no_symbol'}
METHOD PRIVATE FINAL HandleDormantSTATE
VAR_INPUT
END_VAR
VAR_OUTPUT
	xAgain: BOOL;
END_VAR
//判断是否需要重新触发
//IF xExecute AND NOT xDone THEN
IF xExecute THEN
    xBusy:=1;
    eState:=STATE.EXECUTING;
    xAgain:=1;
END_IF

